   DATA[540,19] := 2.0;
   DATA[540,20] := 148.808;
   DATA[540,21] := 155.9344;
   DATA[540,22] := 1.72095;
   DATA[540,23] := 983.6708;
   DATA[540,24] := 2.0;
   DATA[540,25] := 2.0;
   DATA[540,26] := 7.880544;
   DATA[540,27] := 144.9628;
   DATA[540,28] := 263.4581;
   DATA[540,29] := 12.07383;
   DATA[540,30] := 1.73071;
   DATA[540,31] := 1.275778;
   DATA[540,32] := 0.7353967;
   DATA[540,33] := 0.3065689;
   DATA[540,34] := 2.0;
   DATA[540,35] := 251.0254;
   DATA[540,36] := 1.746067;
   DATA[540,37] := 189.8872;
   DATA[540,38] := 0.000128152;
   DATA[540,39] := 1.0;
   DATA[541,0] := 2.535951;
   DATA[541,1] := 533.7197;
   DATA[541,2] := 2.0;
   DATA[541,3] := 2.0;
   DATA[541,4] := 262.1764;
   DATA[541,5] := 8.395475;
   DATA[541,6] := 327.839;
   DATA[541,7] := 2.439753;
   DATA[541,8] := 2.0;
   DATA[541,9] := 2.0;
   DATA[541,10] := 2.0;
   DATA[541,11] := 19.77399;
   DATA[541,12] := 2.214009;
   DATA[541,13] := 980.7582;
   DATA[541,14] := 1.0;
   DATA[541,15] := 2.0;
   DATA[541,16] := 1.0;
   DATA[541,17] := 1.0;
   DATA[541,18] := 1.0;
   DATA[541,19] := 2.0;
   DATA[541,20] := 148.808;
   DATA[541,21] := 155.9344;
   DATA[541,22] := 1.72095;
   DATA[541,23] := 983.7093;
   DATA[541,24] := 2.0;
   DATA[541,25] := 2.0;
   DATA[541,26] := 7.87766;
   DATA[541,27] := 144.9628;
   DATA[541,28] := 263.4581;
   DATA[541,29] := 12.07383;
   DATA[541,30] := 1.730838;
   DATA[541,31] := 1.290893;
   DATA[541,32] := 0.7353967;
   DATA[541,33] := 0.3065689;
   DATA[541,34] := 2.0;
   DATA[541,35] := 251.0254;
   DATA[541,36] := 1.746067;
   DATA[541,37] := 189.8872;
   DATA[541,38] := 0.000128152;
   DATA[541,39] := 1.0;
   DATA[542,0] := 2.51225;
   DATA[542,1] := 534.2693;
   DATA[542,2] := 2.0;
   DATA[542,3] := 2.0;
   DATA[542,4] := 262.1764;
   DATA[542,5] := 8.395475;
   DATA[542,6] := 327.839;
   DATA[542,7] := 2.439753;
   DATA[542,8] := 2.0;
   DATA[542,9] := 2.0;
   DATA[542,10] := 2.0;
   DATA[542,11] := 19.72598;
   DATA[542,12] := 2.214265;
   DATA[542,13] := 980.8783;
   DATA[542,14] := 1.0;
   DATA[542,15] := 2.0;
   DATA[542,16] := 1.0;
   DATA[542,17] := 1.0;
   DATA[542,18] := 1.0;
   DATA[542,19] := 2.0;
   DATA[542,20] := 148.808;
   DATA[542,21] := 155.9344;
   DATA[542,22] := 1.72095;
   DATA[542,23] := 983.9016;
   DATA[542,24] := 2.0;
   DATA[542,25] := 2.0;
   DATA[542,26] := 7.87766;
   DATA[542,27] := 144.9628;
   DATA[542,28] := 263.4581;
   DATA[542,29] := 12.07383;
   DATA[542,30] := 1.730838;
   DATA[542,31] := 1.292686;
   DATA[542,32] := 0.7353967;
   DATA[542,33] := 0.3065689;
   DATA[542,34] := 2.0;
   DATA[542,35] := 251.0254;
   DATA[542,36] := 1.665972;
   DATA[542,37] := 189.759;
   DATA[542,38] := 0.000128152;
   DATA[542,39] := 1.0;
   DATA[543,0] := 2.500721;
   DATA[543,1] := 534.7403;
   DATA[543,2] := 2.0;
   DATA[543,3] := 2.0;
   DATA[543,4] := 262.1764;
   DATA[543,5] := 8.395475;
   DATA[543,6] := 327.839;
   DATA[543,7] := 2.439753;
   DATA[543,8] := 2.0;
   DATA[543,9] := 2.0;
   DATA[543,10] := 2.0;
   DATA[543,11] := 19.72598;
   DATA[543,12] := 2.2126;
   DATA[543,13] := 981.1587;
   DATA[543,14] := 1.0;
   DATA[543,15] := 2.0;
   DATA[543,16] := 1.0;
   DATA[543,17] := 1.0;
   DATA[543,18] := 1.0;
   DATA[543,19] := 2.0;
   DATA[543,20] := 148.808;
   DATA[543,21] := 155.9344;
   DATA[543,22] := 1.718002;
   DATA[543,23] := 984.5552;
   DATA[543,24] := 2.0;
   DATA[543,25] := 2.0;
   DATA[543,26] := 7.87766;
   DATA[543,27] := 144.6296;
   DATA[543,28] := 263.4581;
   DATA[543,29] := 12.07383;
   DATA[543,30] := 1.730838;
   DATA[543,31] := 1.292686;
   DATA[543,32] := 0.7353967;
   DATA[543,33] := 0.3065689;
   DATA[543,34] := 2.0;
   DATA[543,35] := 250.8972;
   DATA[543,36] := 1.665972;
   DATA[543,37] := 189.6469;
   DATA[543,38] := 0.000128152;
   DATA[543,39] := 1.0;
   DATA[544,0] := 2.481504;
   DATA[544,1] := 534.6226;
   DATA[544,2] := 2.0;
   DATA[544,3] := 2.0;
   DATA[544,4] := 262.1764;
   DATA[544,5] := 8.395475;
   DATA[544,6] := 327.839;
   DATA[544,7] := 2.441034;
   DATA[544,8] := 2.0;
   DATA[544,9] := 2.0;
   DATA[544,10] := 2.0;
   DATA[544,11] := 19.68756;
   DATA[544,12] := 2.212087;
   DATA[544,13] := 981.1587;
   DATA[544,14] := 1.0;
   DATA[544,15] := 2.0;
   DATA[544,16] := 1.0;
   DATA[544,17] := 1.0;
   DATA[544,18] := 1.0;
   DATA[544,19] := 2.0;
   DATA[544,20] := 148.808;
   DATA[544,21] := 155.9344;
   DATA[544,22] := 1.715824;
   DATA[544,23] := 984.9782;
   DATA[544,24] := 2.0;
   DATA[544,25] := 2.0;
   DATA[544,26] := 7.87766;
   DATA[544,27] := 144.6296;
   DATA[544,28] := 263.4581;
   DATA[544,29] := 12.07383;
   DATA[544,30] := 1.728531;
   DATA[544,31] := 1.292686;
   DATA[544,32] := 0.7353967;
   DATA[544,33] := 0.3065689;
   DATA[544,34] := 2.0;
   DATA[544,35] := 250.8972;
   DATA[544,36] := 1.665972;
   DATA[544,37] := 189.6469;
   DATA[544,38] := 0.000128152;
   DATA[544,39] := 1.0;
   DATA[545,0] := 2.458764;
   DATA[545,1] := 534.6226;
   DATA[545,2] := 2.0;
   DATA[545,3] := 2.0;
   DATA[545,4] := 262.1764;
   DATA[545,5] := 8.395475;
   DATA[545,6] := 327.839;
   DATA[545,7] := 2.442188;
   DATA[545,8] := 2.0;
   DATA[545,9] := 2.0;
   DATA[545,10] := 2.0;
   DATA[545,11] := 19.68436;
   DATA[545,12] := 2.210037;
   DATA[545,13] := 980.8783;
   DATA[545,14] := 1.0;
   DATA[545,15] := 2.0;
   DATA[545,16] := 1.0;
   DATA[545,17] := 1.0;
   DATA[545,18] := 1.0;
   DATA[545,19] := 2.0;
   DATA[545,20] := 148.808;
   DATA[545,21] := 155.9344;
   DATA[545,22] := 1.715824;
   DATA[545,23] := 985.4396;
   DATA[545,24] := 2.0;
   DATA[545,25] := 2.0;
   DATA[545,26] := 7.87766;
   DATA[545,27] := 144.6296;
   DATA[545,28] := 263.4581;
   DATA[545,29] := 12.07383;
   DATA[545,30] := 1.728531;
   DATA[545,31] := 1.292686;
   DATA[545,32] := 0.7353967;
   DATA[545,33] := 0.3065689;
   DATA[545,34] := 2.0;
   DATA[545,35] := 250.8972;
   DATA[545,36] := 1.665972;
   DATA[545,37] := 189.6469;
   DATA[545,38] := 0.000128152;
   DATA[545,39] := 1.0;
   DATA[546,0] := 2.447875;
   DATA[546,1] := 534.4263;
   DATA[546,2] := 2.0;
   DATA[546,3] := 2.0;
   DATA[546,4] := 262.1764;
   DATA[546,5] := 8.395475;
   DATA[546,6] := 327.839;
   DATA[546,7] := 2.442316;
   DATA[546,8] := 2.0;
   DATA[546,9] := 2.0;
   DATA[546,10] := 2.0;
   DATA[546,11] := 19.67155;
   DATA[546,12] := 2.209397;
   DATA[546,13] := 981.0385;
   DATA[546,14] := 1.0;
   DATA[546,15] := 2.0;
   DATA[546,16] := 1.0;
   DATA[546,17] := 1.0;
   DATA[546,18] := 1.0;
   DATA[546,19] := 2.0;
   DATA[546,20] := 148.808;
   DATA[546,21] := 155.9344;
   DATA[546,22] := 1.71467;
   DATA[546,23] := 985.9011;
   DATA[546,24] := 2.0;
   DATA[546,25] := 2.0;
   DATA[546,26] := 7.87766;
   DATA[546,27] := 144.6296;
   DATA[546,28] := 263.4581;
   DATA[546,29] := 12.07383;
   DATA[546,30] := 1.728531;
   DATA[546,31] := 1.275906;
   DATA[546,32] := 0.7353967;
   DATA[546,33] := 0.3065689;
   DATA[546,34] := 2.0;
   DATA[546,35] := 250.737;
   DATA[546,36] := 1.665972;
   DATA[546,37] := 189.6469;
   DATA[546,38] := 0.000128152;
   DATA[546,39] := 1.0;
   DATA[547,0] := 2.431861;
   DATA[547,1] := 533.7197;
   DATA[547,2] := 2.0;
   DATA[547,3] := 2.0;
   DATA[547,4] := 262.1764;
   DATA[547,5] := 8.395475;
   DATA[547,6] := 327.839;
   DATA[547,7] := 2.442316;
   DATA[547,8] := 2.0;
   DATA[547,9] := 2.0;
   DATA[547,10] := 2.0;
   DATA[547,11] := 19.61073;
   DATA[547,12] := 2.209397;
   DATA[547,13] := 980.8783;
   DATA[547,14] := 1.0;
   DATA[547,15] := 2.0;
   DATA[547,16] := 1.0;
   DATA[547,17] := 1.0;
   DATA[547,18] := 1.0;
   DATA[547,19] := 2.0;
   DATA[547,20] := 148.808;
   DATA[547,21] := 155.9344;
   DATA[547,22] := 1.713389;
   DATA[547,23] := 986.5547;
   DATA[547,24] := 2.0;
   DATA[547,25] := 2.0;
   DATA[547,26] := 7.87766;
   DATA[547,27] := 144.7578;
   DATA[547,28] := 263.4581;
   DATA[547,29] := 12.07383;
   DATA[547,30] := 1.728531;
   DATA[547,31] := 1.27898;
   DATA[547,32] := 0.7353967;
   DATA[547,33] := 0.3086186;
   DATA[547,34] := 2.0;
   DATA[547,35] := 250.721;
   DATA[547,36] := 1.665972;
   DATA[547,37] := 189.5668;
   DATA[547,38] := 0.000128152;
   DATA[547,39] := 1.0;
   DATA[548,0] := 2.422573;
   DATA[548,1] := 533.5627;
   DATA[548,2] := 2.0;
   DATA[548,3] := 2.0;
   DATA[548,4] := 262.1764;
   DATA[548,5] := 8.395475;
   DATA[548,6] := 327.839;
   DATA[548,7] := 2.442316;
   DATA[548,8] := 2.0;
   DATA[548,9] := 2.0;
   DATA[548,10] := 2.0;
   DATA[548,11] := 19.61073;
   DATA[548,12] := 2.209397;
   DATA[548,13] := 980.678;
   DATA[548,14] := 1.0;
   DATA[548,15] := 2.0;
   DATA[548,16] := 1.0;
   DATA[548,17] := 1.0;
   DATA[548,18] := 1.0;
   DATA[548,19] := 2.0;
   DATA[548,20] := 148.808;
   DATA[548,21] := 155.9344;
   DATA[548,22] := 1.713389;
   DATA[548,23] := 986.9777;
   DATA[548,24] := 2.0;
   DATA[548,25] := 2.0;
   DATA[548,26] := 7.87766;
   DATA[548,27] := 144.7578;
   DATA[548,28] := 263.4581;
   DATA[548,29] := 12.07383;
   DATA[548,30] := 1.726865;
   DATA[548,31] := 1.28103;
   DATA[548,32] := 0.7353967;
   DATA[548,33] := 0.3086186;
   DATA[548,34] := 2.0;
   DATA[548,35] := 250.721;
   DATA[548,36] := 1.665972;
   DATA[548,37] := 189.5668;
   DATA[548,38] := 0.000128152;
   DATA[548,39] := 1.0;
   DATA[549,0] := 2.417449;
   DATA[549,1] := 532.5814;
   DATA[549,2] := 2.0;
   DATA[549,3] := 2.0;
   DATA[549,4] := 262.1764;
   DATA[549,5] := 8.395475;
   DATA[549,6] := 327.839;
   DATA[549,7] := 2.442316;
   DATA[549,8] := 2.0;
   DATA[549,9] := 2.0;
   DATA[549,10] := 2.0;
   DATA[549,11] := 19.61073;
   DATA[549,12] := 2.205682;
   DATA[549,13] := 981.4791;
   DATA[549,14] := 1.0;
   DATA[549,15] := 2.0;
   DATA[549,16] := 1.0;
   DATA[549,17] := 1.0;
   DATA[549,18] := 1.0;
   DATA[549,19] := 2.0;
   DATA[549,20] := 148.808;
   DATA[549,21] := 155.9344;
   DATA[549,22] := 1.714029;
   DATA[549,23] := 987.7083;
   DATA[549,24] := 2.0;
   DATA[549,25] := 2.0;
   DATA[549,26] := 7.87766;
   DATA[549,27] := 144.7578;
   DATA[549,28] := 263.4581;
   DATA[549,29] := 12.07383;
   DATA[549,30] := 1.726865;
   DATA[549,31] := 1.285513;
   DATA[549,32] := 0.7353967;
   DATA[549,33] := 0.3075937;
   DATA[549,34] := 2.0;
   DATA[549,35] := 250.721;
   DATA[549,36] := 1.665972;
   DATA[549,37] := 189.5668;
   DATA[549,38] := 0.000128152;
   DATA[549,39] := 1.0;
   DATA[550,0] := 2.417449;
   DATA[550,1] := 532.5814;
   DATA[550,2] := 2.0;
   DATA[550,3] := 2.0;
   DATA[550,4] := 262.1764;
   DATA[550,5] := 8.395475;
   DATA[550,6] := 327.839;
   DATA[550,7] := 2.442316;
   DATA[550,8] := 2.0;
   DATA[550,9] := 2.0;
   DATA[550,10] := 2.0;
   DATA[550,11] := 19.61073;
   DATA[550,12] := 2.205682;
   DATA[550,13] := 981.4791;
   DATA[550,14] := 1.0;
   DATA[550,15] := 2.0;
   DATA[550,16] := 1.0;
   DATA[550,17] := 1.0;
   DATA[550,18] := 1.0;
   DATA[550,19] := 2.0;
   DATA[550,20] := 148.808;
   DATA[550,21] := 155.9344;
   DATA[550,22] := 1.714029;
   DATA[550,23] := 987.7083;
   DATA[550,24] := 2.0;
   DATA[550,25] := 2.0;
   DATA[550,26] := 7.87766;
   DATA[550,27] := 144.7578;
   DATA[550,28] := 263.4581;
   DATA[550,29] := 12.07383;
   DATA[550,30] := 1.726865;
   DATA[550,31] := 1.285513;
   DATA[550,32] := 0.7353967;
   DATA[550,33] := 0.3075937;
   DATA[550,34] := 2.0;
   DATA[550,35] := 250.721;
   DATA[550,36] := 1.665972;
   DATA[550,37] := 189.5668;
   DATA[550,38] := 0.000128152;
   DATA[550,39] := 1.0;
   DATA[551,0] := 2.423534;
   DATA[551,1] := 532.2674;
   DATA[551,2] := 2.0;
   DATA[551,3] := 2.0;
   DATA[551,4] := 262.1764;
   DATA[551,5] := 8.395475;
   DATA[551,6] := 327.839;
   DATA[551,7] := 2.441547;
   DATA[551,8] := 2.0;
   DATA[551,9] := 2.0;
   DATA[551,10] := 2.0;
   DATA[551,11] := 19.61073;
   DATA[551,12] := 2.205682;
   DATA[551,13] := 981.5593;
   DATA[551,14] := 1.0;
   DATA[551,15] := 2.0;
   DATA[551,16] := 1.0;
   DATA[551,17] := 1.0;
   DATA[551,18] := 1.0;
   DATA[551,19] := 2.0;
   DATA[551,20] := 148.808;
   DATA[551,21] := 155.9344;
   DATA[551,22] := 1.716849;
   DATA[551,23] := 988.0159;
   DATA[551,24] := 2.0;
   DATA[551,25] := 2.0;
   DATA[551,26] := 7.87766;
   DATA[551,27] := 144.7578;
   DATA[551,28] := 263.4581;
   DATA[551,29] := 12.07383;
   DATA[551,30] := 1.726865;
   DATA[551,31] := 1.291405;
   DATA[551,32] := 0.7353967;
   DATA[551,33] := 0.3065689;
   DATA[551,34] := 2.0;
   DATA[551,35] := 250.9773;
   DATA[551,36] := 1.665972;
   DATA[551,37] := 189.5668;
   DATA[551,38] := 0.000128152;
   DATA[551,39] := 1.0;
   DATA[552,0] := 2.455241;
   DATA[552,1] := 531.3253;
   DATA[552,2] := 2.0;
   DATA[552,3] := 2.0;
   DATA[552,4] := 262.1764;
   DATA[552,5] := 8.395475;
   DATA[552,6] := 327.839;
   DATA[552,7] := 2.441547;
   DATA[552,8] := 2.0;
   DATA[552,9] := 2.0;
   DATA[552,10] := 2.0;
   DATA[552,11] := 19.67155;
   DATA[552,12] := 2.208884;
   DATA[552,13] := 981.8796;
   DATA[552,14] := 1.0;
   DATA[552,15] := 2.0;
   DATA[552,16] := 1.0;
   DATA[552,17] := 1.0;
   DATA[552,18] := 1.0;
   DATA[552,19] := 2.0;
   DATA[552,20] := 148.808;
   DATA[552,21] := 155.9344;
   DATA[552,22] := 1.718771;
   DATA[552,23] := 987.939;
   DATA[552,24] := 2.0;
   DATA[552,25] := 2.0;
   DATA[552,26] := 7.87766;
   DATA[552,27] := 144.7578;
   DATA[552,28] := 263.4581;
   DATA[552,29] := 12.07383;
   DATA[552,30] := 1.726865;
   DATA[552,31] := 1.28436;
   DATA[552,32] := 0.7377012;
   DATA[552,33] := 0.3062486;
   DATA[552,34] := 2.0;
   DATA[552,35] := 251.0574;
   DATA[552,36] := 1.778105;
   DATA[552,37] := 189.743;
   DATA[552,38] := 0.000128152;
   DATA[552,39] := 1.0;
   DATA[553,0] := 2.494315;
   DATA[553,1] := 530.7758;
   DATA[553,2] := 2.0;
   DATA[553,3] := 2.0;
   DATA[553,4] := 262.1764;
   DATA[553,5] := 8.395475;
   DATA[553,6] := 327.839;
   DATA[553,7] := 2.441547;
   DATA[553,8] := 2.0;
   DATA[553,9] := 2.0;
   DATA[553,10] := 2.0;
   DATA[553,11] := 19.70037;
   DATA[553,12] := 2.208884;
   DATA[553,13] := 981.7595;
   DATA[553,14] := 1.0;
   DATA[553,15] := 2.0;
   DATA[553,16] := 1.0;
   DATA[553,17] := 1.0;
   DATA[553,18] := 1.0;
   DATA[553,19] := 2.0;
   DATA[553,20] := 148.808;
   DATA[553,21] := 155.9344;
   DATA[553,22] := 1.719924;
   DATA[553,23] := 988.2081;
   DATA[553,24] := 2.0;
   DATA[553,25] := 2.0;
   DATA[553,26] := 7.878942;
   DATA[553,27] := 144.7578;
   DATA[553,28] := 263.4581;
   DATA[553,29] := 12.07383;
   DATA[553,30] := 1.726865;
   DATA[553,31] := 1.281542;
   DATA[553,32] := 0.7377012;
   DATA[553,33] := 0.3062486;
   DATA[553,34] := 2.0;
   DATA[553,35] := 251.2016;
   DATA[553,36] := 1.778105;
   DATA[553,37] := 189.8231;
   DATA[553,38] := 0.000128152;
   DATA[553,39] := 1.0;
   DATA[554,0] := 2.54652;
   DATA[554,1] := 529.7159;
   DATA[554,2] := 2.0;
   DATA[554,3] := 2.0;
   DATA[554,4] := 262.1764;
   DATA[554,5] := 8.395475;
   DATA[554,6] := 327.839;
   DATA[554,7] := 2.441547;
   DATA[554,8] := 2.0;
   DATA[554,9] := 2.0;
   DATA[554,10] := 2.0;
   DATA[554,11] := 19.71637;
   DATA[554,12] := 2.208884;
   DATA[554,13] := 981.5593;
   DATA[554,14] := 1.0;
   DATA[554,15] := 2.0;
   DATA[554,16] := 1.0;
   DATA[554,17] := 1.0;
   DATA[554,18] := 1.0;
   DATA[554,19] := 2.0;
   DATA[554,20] := 148.808;
   DATA[554,21] := 155.9344;
   DATA[554,22] := 1.723256;
   DATA[554,23] := 988.5157;
   DATA[554,24] := 2.0;
   DATA[554,25] := 2.0;
   DATA[554,26] := 7.880544;
   DATA[554,27] := 144.7578;
   DATA[554,28] := 263.4581;
   DATA[554,29] := 12.07383;
   DATA[554,30] := 1.726865;
   DATA[554,31] := 1.281542;
   DATA[554,32] := 0.7377012;
   DATA[554,33] := 0.3062486;
   DATA[554,34] := 2.0;
   DATA[554,35] := 251.2977;
   DATA[554,36] := 1.778105;
   DATA[554,37] := 189.9833;
   DATA[554,38] := 0.000128152;
   DATA[554,39] := 1.0;
   DATA[555,0] := 2.570541;
   DATA[555,1] := 529.3627;
   DATA[555,2] := 2.0;
   DATA[555,3] := 2.0;
   DATA[555,4] := 262.1764;
   DATA[555,5] := 8.395475;
   DATA[555,6] := 327.839;
   DATA[555,7] := 2.441547;
   DATA[555,8] := 2.0;
   DATA[555,9] := 2.0;
   DATA[555,10] := 2.0;
   DATA[555,11] := 19.75159;
   DATA[555,12] := 2.208884;
   DATA[555,13] := 981.2789;
   DATA[555,14] := 1.0;
   DATA[555,15] := 2.0;
   DATA[555,16] := 1.0;
   DATA[555,17] := 1.0;
   DATA[555,18] := 1.0;
   DATA[555,19] := 2.0;
   DATA[555,20] := 148.808;
   DATA[555,21] := 155.9344;
   DATA[555,22] := 1.724153;
   DATA[555,23] := 988.4388;
   DATA[555,24] := 2.0;
   DATA[555,25] := 2.0;
   DATA[555,26] := 7.880544;
   DATA[555,27] := 144.7578;
   DATA[555,28] := 263.4581;
   DATA[555,29] := 12.07383;
   DATA[555,30] := 1.728019;
   DATA[555,31] := 1.288715;
   DATA[555,32] := 0.7379573;
   DATA[555,33] := 0.3062486;
   DATA[555,34] := 2.0;
   DATA[555,35] := 251.2977;
   DATA[555,36] := 1.778105;
   DATA[555,37] := 190.0474;
   DATA[555,38] := 0.000128152;
   DATA[555,39] := 1.0;
   DATA[556,0] := 2.61634;
   DATA[556,1] := 528.5776;
   DATA[556,2] := 2.0;
   DATA[556,3] := 2.0;
   DATA[556,4] := 262.1764;
   DATA[556,5] := 8.395475;
   DATA[556,6] := 327.839;
   DATA[556,7] := 2.441547;
   DATA[556,8] := 2.0;
   DATA[556,9] := 2.0;
   DATA[556,10] := 2.0;
   DATA[556,11] := 19.79;
   DATA[556,12] := 2.208372;
   DATA[556,13] := 981.1987;
   DATA[556,14] := 1.0;
   DATA[556,15] := 2.0;
   DATA[556,16] := 1.0;
   DATA[556,17] := 1.0;
   DATA[556,18] := 1.0;
   DATA[556,19] := 2.0;
   DATA[556,20] := 148.808;
   DATA[556,21] := 156.0369;
   DATA[556,22] := 1.724153;
   DATA[556,23] := 989.0156;
   DATA[556,24] := 2.0;
   DATA[556,25] := 2.0;
   DATA[556,26] := 7.880544;
   DATA[556,27] := 144.7578;
   DATA[556,28] := 263.4581;
   DATA[556,29] := 12.07383;
   DATA[556,30] := 1.729172;
   DATA[556,31] := 1.292558;
   DATA[556,32] := 0.7357808;
   DATA[556,33] := 0.3066329;
   DATA[556,34] := 2.0;
   DATA[556,35] := 251.2977;
   DATA[556,36] := 1.778105;
   DATA[556,37] := 190.0474;
   DATA[556,38] := 0.000128152;
   DATA[556,39] := 1.0;
   DATA[557,0] := 2.641322;
   DATA[557,1] := 528.4599;
   DATA[557,2] := 2.0;
   DATA[557,3] := 2.0;
   DATA[557,4] := 262.1764;
   DATA[557,5] := 8.395475;
   DATA[557,6] := 327.9159;
   DATA[557,7] := 2.441162;
   DATA[557,8] := 2.0;
   DATA[557,9] := 2.0;
   DATA[557,10] := 2.0;
   DATA[557,11] := 19.80601;
   DATA[557,12] := 2.208372;
   DATA[557,13] := 981.4391;
   DATA[557,14] := 1.0;
   DATA[557,15] := 2.0;
   DATA[557,16] := 1.0;
   DATA[557,17] := 1.0;
   DATA[557,18] := 1.0;
   DATA[557,19] := 2.0;
   DATA[557,20] := 148.808;
   DATA[557,21] := 156.0369;
   DATA[557,22] := 1.724153;
   DATA[557,23] := 988.708;
   DATA[557,24] := 2.0;
   DATA[557,25] := 2.0;
   DATA[557,26] := 7.880544;
   DATA[557,27] := 144.7578;
   DATA[557,28] := 263.4581;
   DATA[557,29] := 12.07383;
   DATA[557,30] := 1.729172;
   DATA[557,31] := 1.292558;
   DATA[557,32] := 0.7357808;
   DATA[557,33] := 0.3066329;
   DATA[557,34] := 2.0;
   DATA[557,35] := 251.2977;
   DATA[557,36] := 1.778105;
   DATA[557,37] := 190.0474;
   DATA[557,38] := 0.000128152;
   DATA[557,39] := 1.0;
   DATA[558,0] := 2.672389;
   DATA[558,1] := 528.8132;
   DATA[558,2] := 2.0;
   DATA[558,3] := 2.0;
   DATA[558,4] := 262.1764;
   DATA[558,5] := 8.395475;
   DATA[558,6] := 327.9159;
   DATA[558,7] := 2.440265;
   DATA[558,8] := 2.0;
   DATA[558,9] := 2.0;
   DATA[558,10] := 2.0;
   DATA[558,11] := 19.80601;
   DATA[558,12] := 2.210806;
   DATA[558,13] := 981.7996;
   DATA[558,14] := 1.0;
   DATA[558,15] := 2.0;
   DATA[558,16] := 1.0;
   DATA[558,17] := 1.0;
   DATA[558,18] := 1.0;
   DATA[558,19] := 2.0;
   DATA[558,20] := 148.808;
   DATA[558,21] := 156.0369;
   DATA[558,22] := 1.724153;
   DATA[558,23] := 988.9003;
   DATA[558,24] := 2.0;
   DATA[558,25] := 2.0;
   DATA[558,26] := 7.880544;
   DATA[558,27] := 144.7578;
   DATA[558,28] := 263.4581;
   DATA[558,29] := 12.07383;
   DATA[558,30] := 1.729172;
   DATA[558,31] := 1.292174;
   DATA[558,32] := 0.7357808;
   DATA[558,33] := 0.3074656;
   DATA[558,34] := 2.0;
   DATA[558,35] := 251.2977;
   DATA[558,36] := 1.778105;
   DATA[558,37] := 190.0474;
   DATA[558,38] := 0.000128152;
   DATA[558,39] := 1.0;
   DATA[559,0] := 2.674951;
   DATA[559,1] := 528.7739;
   DATA[559,2] := 2.0;
   DATA[559,3] := 2.0;
   DATA[559,4] := 262.1764;
   DATA[559,5] := 8.395475;
   DATA[559,6] := 327.9159;
   DATA[559,7] := 2.440265;
   DATA[559,8] := 2.0;
   DATA[559,9] := 2.0;
   DATA[559,10] := 2.0;
   DATA[559,11] := 19.73238;
   DATA[559,12] := 2.211959;
   DATA[559,13] := 981.5993;
   DATA[559,14] := 1.0;
   DATA[559,15] := 2.0;
   DATA[559,16] := 1.0;
   DATA[559,17] := 1.0;
   DATA[559,18] := 1.0;
   DATA[559,19] := 2.0;
   DATA[559,20] := 148.808;
   DATA[559,21] := 156.0369;
   DATA[559,22] := 1.723641;
   DATA[559,23] := 988.6696;
   DATA[559,24] := 2.0;
   DATA[559,25] := 2.0;
   DATA[559,26] := 7.880544;
   DATA[559,27] := 144.7578;
   DATA[559,28] := 263.4581;
   DATA[559,29] := 12.07383;
   DATA[559,30] := 1.730838;
   DATA[559,31] := 1.283079;
   DATA[559,32] := 0.7353967;
   DATA[559,33] := 0.3080421;
   DATA[559,34] := 2.0;
   DATA[559,35] := 251.2977;
   DATA[559,36] := 1.746067;
   DATA[559,37] := 190.0474;
   DATA[559,38] := 0.000128152;
   DATA[559,39] := 1.0;
   DATA[560,0] := 2.643244;
   DATA[560,1] := 529.6375;
   DATA[560,2] := 2.0;
   DATA[560,3] := 2.0;
   DATA[560,4] := 262.1764;
   DATA[560,5] := 8.395475;
   DATA[560,6] := 327.9159;
   DATA[560,7] := 2.4427;
   DATA[560,8] := 2.0;
   DATA[560,9] := 2.0;
   DATA[560,10] := 2.0;
   DATA[560,11] := 19.69076;
   DATA[560,12] := 2.211959;
   DATA[560,13] := 981.1987;
   DATA[560,14] := 1.0;
   DATA[560,15] := 2.0;
   DATA[560,16] := 1.0;
   DATA[560,17] := 1.0;
   DATA[560,18] := 1.0;
   DATA[560,19] := 2.0;
   DATA[560,20] := 148.808;
   DATA[560,21] := 156.0369;
   DATA[560,22] := 1.722487;
   DATA[560,23] := 988.6696;
   DATA[560,24] := 2.0;
   DATA[560,25] := 2.0;
   DATA[560,26] := 7.880544;
   DATA[560,27] := 144.7578;
   DATA[560,28] := 263.4581;
   DATA[560,29] := 12.07383;
   DATA[560,30] := 1.731479;
   DATA[560,31] := 1.287306;
   DATA[560,32] := 0.7353967;
   DATA[560,33] := 0.3080421;
   DATA[560,34] := 2.0;
   DATA[560,35] := 251.2977;
   DATA[560,36] := 1.746067;
   DATA[560,37] := 190.0474;
   DATA[560,38] := 0.000128152;
   DATA[560,39] := 1.0;
   DATA[561,0] := 2.621785;
   DATA[561,1] := 530.344;
   DATA[561,2] := 2.0;
   DATA[561,3] := 2.0;
   DATA[561,4] := 262.1764;
   DATA[561,5] := 8.395475;
   DATA[561,6] := 327.9159;
   DATA[561,7] := 2.4427;
   DATA[561,8] := 2.0;
   DATA[561,9] := 2.0;
   DATA[561,10] := 2.0;
   DATA[561,11] := 19.66835;
   DATA[561,12] := 2.211959;
   DATA[561,13] := 981.4791;
   DATA[561,14] := 1.0;
   DATA[561,15] := 2.0;
   DATA[561,16] := 1.0;
   DATA[561,17] := 1.0;
   DATA[561,18] := 1.0;
   DATA[561,19] := 2.0;
   DATA[561,20] := 148.808;
   DATA[561,21] := 156.0369;
   DATA[561,22] := 1.72159;
   DATA[561,23] := 988.7465;
   DATA[561,24] := 2.0;
   DATA[561,25] := 2.0;
   DATA[561,26] := 7.880544;
   DATA[561,27] := 144.7578;
   DATA[561,28] := 263.4261;
   DATA[561,29] := 12.07383;
   DATA[561,30] := 1.731479;
   DATA[561,31] := 1.274625;
   DATA[561,32] := 0.7353967;
   DATA[561,33] := 0.3087468;
   DATA[561,34] := 2.0;
   DATA[561,35] := 251.2977;
   DATA[561,36] := 1.746067;
   DATA[561,37] := 190.0474;
   DATA[561,38] := 0.000128152;
   DATA[561,39] := 1.0;
   DATA[562,0] := 2.61634;
   DATA[562,1] := 531.9534;
   DATA[562,2] := 2.0;
   DATA[562,3] := 2.0;
   DATA[562,4] := 262.1764;
   DATA[562,5] := 8.395475;
   DATA[562,6] := 327.9159;
   DATA[562,7] := 2.4427;
   DATA[562,8] := 2.0;
   DATA[562,9] := 2.0;
   DATA[562,10] := 2.0;
   DATA[562,11] := 19.66835;
   DATA[562,12] := 2.214906;
   DATA[562,13] := 981.4391;
   DATA[562,14] := 1.0;
   DATA[562,15] := 2.0;
   DATA[562,16] := 1.0;
   DATA[562,17] := 1.0;
   DATA[562,18] := 1.0;
   DATA[562,19] := 2.0;
   DATA[562,20] := 148.808;
   DATA[562,21] := 156.0369;
   DATA[562,22] := 1.718515;
   DATA[562,23] := 989.0925;
   DATA[562,24] := 2.0;
   DATA[562,25] := 2.0;
   DATA[562,26] := 7.880544;
   DATA[562,27] := 144.7578;
   DATA[562,28] := 263.4261;
   DATA[562,29] := 12.07383;
   DATA[562,30] := 1.731479;
   DATA[562,31] := 1.261432;
   DATA[562,32] := 0.7353967;
   DATA[562,33] := 0.3068891;
   DATA[562,34] := 2.0;
   DATA[562,35] := 251.0734;
   DATA[562,36] := 1.746067;
   DATA[562,37] := 189.727;
   DATA[562,38] := 0.000128152;
   DATA[562,39] := 1.0;
   DATA[563,0] := 2.6157;
   DATA[563,1] := 532.5422;
   DATA[563,2] := 2.0;
   DATA[563,3] := 2.0;
   DATA[563,4] := 262.1764;
   DATA[563,5] := 8.395155;
   DATA[563,6] := 327.9159;
   DATA[563,7] := 2.4427;
   DATA[563,8] := 2.0;
   DATA[563,9] := 2.0;
   DATA[563,10] := 2.0;
   DATA[563,11] := 19.66835;
   DATA[563,12] := 2.214906;
   DATA[563,13] := 981.5593;
   DATA[563,14] := 1.0;
   DATA[563,15] := 2.0;
   DATA[563,16] := 1.0;
   DATA[563,17] := 1.0;
   DATA[563,18] := 1.0;
   DATA[563,19] := 2.0;
   DATA[563,20] := 148.808;
   DATA[563,21] := 156.0369;
   DATA[563,22] := 1.718515;
   DATA[563,23] := 988.708;
   DATA[563,24] := 2.0;
   DATA[563,25] := 2.0;
   DATA[563,26] := 7.880544;
   DATA[563,27] := 144.7578;
   DATA[563,28] := 263.4261;
   DATA[563,29] := 12.07383;
   DATA[563,30] := 1.731479;
   DATA[563,31] := 1.25554;
   DATA[563,32] := 0.7353967;
   DATA[563,33] := 0.3066329;
   DATA[563,34] := 2.0;
   DATA[563,35] := 251.0734;
   DATA[563,36] := 1.746067;
   DATA[563,37] := 189.727;
   DATA[563,38] := 0.000128152;
   DATA[563,39] := 1.0;
   DATA[564,0] := 2.593601;
   DATA[564,1] := 532.8954;
   DATA[564,2] := 2.0;
   DATA[564,3] := 2.0;
   DATA[564,4] := 262.1764;
   DATA[564,5] := 8.394835;
   DATA[564,6] := 327.9159;
   DATA[564,7] := 2.444879;
   DATA[564,8] := 2.0;
   DATA[564,9] := 2.0;
   DATA[564,10] := 2.0;
   DATA[564,11] := 19.66835;
   DATA[564,12] := 2.21324;
   DATA[564,13] := 980.8383;
   DATA[564,14] := 1.0;
   DATA[564,15] := 2.0;
   DATA[564,16] := 1.0;
   DATA[564,17] := 1.0;
   DATA[564,18] := 1.0;
   DATA[564,19] := 2.0;
   DATA[564,20] := 148.808;
   DATA[564,21] := 156.0369;
   DATA[564,22] := 1.718515;
   DATA[564,23] := 989.0925;
   DATA[564,24] := 2.0;
   DATA[564,25] := 2.0;
   DATA[564,26] := 7.880544;
   DATA[564,27] := 144.7578;
   DATA[564,28] := 263.4261;
   DATA[564,29] := 12.07383;
   DATA[564,30] := 1.7293;
   DATA[564,31] := 1.254643;
   DATA[564,32] := 0.7353967;
   DATA[564,33] := 0.3065048;
   DATA[564,34] := 2.0;
   DATA[564,35] := 250.9773;
   DATA[564,36] := 1.746067;
   DATA[564,37] := 189.727;
   DATA[564,38] := 0.000128152;
   DATA[564,39] := 1.0;
   DATA[565,0] := 2.572142;
   DATA[565,1] := 532.9739;
   DATA[565,2] := 2.0;
   DATA[565,3] := 2.0;
   DATA[565,4] := 262.1764;
   DATA[565,5] := 8.394835;
   DATA[565,6] := 327.9159;
   DATA[565,7] := 2.444879;
   DATA[565,8] := 2.0;
   DATA[565,9] := 2.0;
   DATA[565,10] := 2.0;
   DATA[565,11] := 19.67796;
   DATA[565,12] := 2.21324;
   DATA[565,13] := 981.1587;
   DATA[565,14] := 1.0;
   DATA[565,15] := 2.0;
   DATA[565,16] := 1.0;
   DATA[565,17] := 1.0;
   DATA[565,18] := 1.0;
   DATA[565,19] := 2.0;
   DATA[565,20] := 148.808;
   DATA[565,21] := 156.0369;
   DATA[565,22] := 1.718515;
   DATA[565,23] := 988.9387;
   DATA[565,24] := 2.0;
   DATA[565,25] := 2.0;
   DATA[565,26] := 7.880544;
   DATA[565,27] := 144.7578;
   DATA[565,28] := 263.4261;
   DATA[565,29] := 12.07383;
   DATA[565,30] := 1.7293;
   DATA[565,31] := 1.268989;
   DATA[565,32] := 0.7353967;
   DATA[565,33] := 0.3065048;
   DATA[565,34] := 2.0;
   DATA[565,35] := 250.9132;
   DATA[565,36] := 1.746067;
   DATA[565,37] := 189.5988;
   DATA[565,38] := 0.000128152;
   DATA[565,39] := 1.0;
   DATA[566,0] := 2.560933;
   DATA[566,1] := 532.8562;
   DATA[566,2] := 2.0;
   DATA[566,3] := 2.0;
   DATA[566,4] := 262.1764;
   DATA[566,5] := 8.394835;
   DATA[566,6] := 327.9159;
   DATA[566,7] := 2.444879;
   DATA[566,8] := 2.0;
   DATA[566,9] := 2.0;
   DATA[566,10] := 2.0;
   DATA[566,11] := 19.67796;
   DATA[566,12] := 2.21324;
   DATA[566,13] := 981.1987;
   DATA[566,14] := 1.0;
   DATA[566,15] := 2.0;
   DATA[566,16] := 1.0;
   DATA[566,17] := 1.0;
   DATA[566,18] := 1.0;
   DATA[566,19] := 2.0;
   DATA[566,20] := 148.808;
   DATA[566,21] := 156.0369;
   DATA[566,22] := 1.717105;
   DATA[566,23] := 988.4773;
   DATA[566,24] := 2.0;
   DATA[566,25] := 2.0;
   DATA[566,26] := 7.880544;
   DATA[566,27] := 144.7578;
   DATA[566,28] := 263.4261;
   DATA[566,29] := 12.07383;
   DATA[566,30] := 1.726096;
   DATA[566,31] := 1.271039;
   DATA[566,32] := 0.736421;
   DATA[566,33] := 0.3065048;
   DATA[566,34] := 2.0;
   DATA[566,35] := 250.5928;
   DATA[566,36] := 1.665972;
   DATA[566,37] := 189.5347;
   DATA[566,38] := 0.000128152;
   DATA[566,39] := 1.0;
   DATA[567,0] := 2.542036;
   DATA[567,1] := 532.7384;
   DATA[567,2] := 2.0;
   DATA[567,3] := 2.0;
   DATA[567,4] := 262.1764;
   DATA[567,5] := 8.394835;
   DATA[567,6] := 327.9159;
   DATA[567,7] := 2.442444;
   DATA[567,8] := 2.0;
   DATA[567,9] := 2.0;
   DATA[567,10] := 2.0;
   DATA[567,11] := 19.67796;
   DATA[567,12] := 2.21324;
   DATA[567,13] := 981.1587;
   DATA[567,14] := 1.0;
   DATA[567,15] := 2.0;
   DATA[567,16] := 1.0;
   DATA[567,17] := 1.0;
   DATA[567,18] := 1.0;
   DATA[567,19] := 2.0;
   DATA[567,20] := 148.808;
   DATA[567,21] := 156.0369;
   DATA[567,22] := 1.716592;
   DATA[567,23] := 989.0541;
   DATA[567,24] := 2.0;
   DATA[567,25] := 2.0;
   DATA[567,26] := 7.880544;
   DATA[567,27] := 144.8859;
   DATA[567,28] := 263.4261;
   DATA[567,29] := 12.07383;
   DATA[567,30] := 1.726096;
   DATA[567,31] := 1.280261;
   DATA[567,32] := 0.7370611;
   DATA[567,33] := 0.3065048;
   DATA[567,34] := 2.0;
   DATA[567,35] := 250.5928;
   DATA[567,36] := 1.665972;
   DATA[567,37] := 189.5027;
   DATA[567,38] := 0.000128152;
   DATA[567,39] := 1.0;
   DATA[568,0] := 2.530506;
   DATA[568,1] := 532.4637;
   DATA[568,2] := 2.0;
   DATA[568,3] := 2.0;
   DATA[568,4] := 262.1764;
   DATA[568,5] := 8.394835;
   DATA[568,6] := 327.9159;
   DATA[568,7] := 2.441162;
   DATA[568,8] := 2.0;
   DATA[568,9] := 2.0;
   DATA[568,10] := 2.0;
   DATA[568,11] := 19.63954;
   DATA[568,12] := 2.211318;
   DATA[568,13] := 980.9985;
   DATA[568,14] := 1.0;
   DATA[568,15] := 2.0;
   DATA[568,16] := 1.0;
   DATA[568,17] := 1.0;
   DATA[568,18] := 1.0;
   DATA[568,19] := 2.0;
   DATA[568,20] := 148.808;
   DATA[568,21] := 156.0369;
   DATA[568,22] := 1.716592;
   DATA[568,23] := 988.708;
   DATA[568,24] := 2.0;
   DATA[568,25] := 2.0;
   DATA[568,26] := 7.880544;
   DATA[568,27] := 144.9116;
   DATA[568,28] := 263.4261;
   DATA[568,29] := 12.07383;
   DATA[568,30] := 1.726096;
   DATA[568,31] := 1.290124;
   DATA[568,32] := 0.7370611;
   DATA[568,33] := 0.3083624;
   DATA[568,34] := 2.0;
   DATA[568,35] := 250.5928;
   DATA[568,36] := 1.665972;
   DATA[568,37] := 189.5027;
   DATA[568,38] := 0.000128152;
   DATA[568,39] := 1.0;
   DATA[569,0] := 2.510649;
   DATA[569,1] := 532.2674;
   DATA[569,2] := 2.0;
   DATA[569,3] := 2.0;
   DATA[569,4] := 262.1764;
   DATA[569,5] := 8.394835;
   DATA[569,6] := 327.9159;
   DATA[569,7] := 2.440521;
   DATA[569,8] := 2.0;
   DATA[569,9] := 2.0;
   DATA[569,10] := 2.0;
   DATA[569,11] := 19.63954;
   DATA[569,12] := 2.210294;
   DATA[569,13] := 980.638;
   DATA[569,14] := 1.0;
   DATA[569,15] := 2.0;
   DATA[569,16] := 1.0;
   DATA[569,17] := 1.0;
   DATA[569,18] := 1.0;
   DATA[569,19] := 2.0;
   DATA[569,20] := 148.808;
   DATA[569,21] := 156.0369;
   DATA[569,22] := 1.717746;
   DATA[569,23] := 988.8618;
   DATA[569,24] := 2.0;
   DATA[569,25] := 2.0;
   DATA[569,26] := 7.880544;
   DATA[569,27] := 144.9116;
   DATA[569,28] := 263.4261;
   DATA[569,29] := 12.07383;
   DATA[569,30] := 1.726096;
   DATA[569,31] := 1.291277;
   DATA[569,32] := 0.7370611;
   DATA[569,33] := 0.3083624;
   DATA[569,34] := 2.0;
   DATA[569,35] := 250.8171;
   DATA[569,36] := 1.665972;
   DATA[569,37] := 189.5027;
   DATA[569,38] := 0.000128152;
   DATA[569,39] := 1.0;
   DATA[570,0] := 2.498799;
   DATA[570,1] := 532.3459;
   DATA[570,2] := 2.0;
   DATA[570,3] := 2.0;
   DATA[570,4] := 262.1764;
   DATA[570,5] := 8.394835;
   DATA[570,6] := 327.9159;
   DATA[570,7] := 2.439881;
   DATA[570,8] := 2.0;
   DATA[570,9] := 2.0;
   DATA[570,10] := 2.0;
   DATA[570,11] := 19.63954;
   DATA[570,12] := 2.210294;
   DATA[570,13] := 980.598;
   DATA[570,14] := 1.0;
   DATA[570,15] := 2.0;
   DATA[570,16] := 1.0;
   DATA[570,17] := 1.0;
   DATA[570,18] := 1.0;
   DATA[570,19] := 2.0;
   DATA[570,20] := 148.808;
   DATA[570,21] := 156.0369;
   DATA[570,22] := 1.717746;
   DATA[570,23] := 988.8618;
   DATA[570,24] := 2.0;
   DATA[570,25] := 2.0;
   DATA[570,26] := 7.880544;
   DATA[570,27] := 144.9116;
   DATA[570,28] := 263.4261;
   DATA[570,29] := 12.07383;
   DATA[570,30] := 1.726096;
   DATA[570,31] := 1.286025;
   DATA[570,32] := 0.7359089;
   DATA[570,33] := 0.3083624;
   DATA[570,34] := 2.0;
   DATA[570,35] := 250.8652;
   DATA[570,36] := 1.665972;
   DATA[570,37] := 189.5027;
   DATA[570,38] := 0.000128152;
   DATA[570,39] := 1.0;
   DATA[571,0] := 2.484066;
   DATA[571,1] := 532.1497;
   DATA[571,2] := 2.0;
   DATA[571,3] := 2.0;
   DATA[571,4] := 262.1764;
   DATA[571,5] := 8.394835;
   DATA[571,6] := 327.9159;
   DATA[571,7] := 2.439881;
   DATA[571,8] := 2.0;
   DATA[571,9] := 2.0;
   DATA[571,10] := 2.0;
   DATA[571,11] := 19.65875;
   DATA[571,12] := 2.214777;
   DATA[571,13] := 980.638;
   DATA[571,14] := 1.0;
   DATA[571,15] := 2.0;
   DATA[571,16] := 1.0;
   DATA[571,17] := 1.0;
   DATA[571,18] := 1.0;
   DATA[571,19] := 2.0;
   DATA[571,20] := 148.808;
   DATA[571,21] := 156.0369;
   DATA[571,22] := 1.717746;
   DATA[571,23] := 989.4386;
   DATA[571,24] := 2.0;
   DATA[571,25] := 2.0;
   DATA[571,26] := 7.880544;
   DATA[571,27] := 144.9116;
   DATA[571,28] := 263.4261;
   DATA[571,29] := 12.07383;
   DATA[571,30] := 1.726096;
   DATA[571,31] := 1.287947;
   DATA[571,32] := 0.7347566;
   DATA[571,33] := 0.3083624;
   DATA[571,34] := 2.0;
   DATA[571,35] := 250.9453;
   DATA[571,36] := 1.665972;
   DATA[571,37] := 189.743;
   DATA[571,38] := 0.000128152;
   DATA[571,39] := 1.0;
   DATA[572,0] := 2.475098;
   DATA[572,1] := 532.0711;
   DATA[572,2] := 2.0;
   DATA[572,3] := 2.0;
   DATA[572,4] := 262.1764;
   DATA[572,5] := 8.394835;
   DATA[572,6] := 327.9159;
   DATA[572,7] := 2.439881;
   DATA[572,8] := 2.0;
   DATA[572,9] := 2.0;
   DATA[572,10] := 2.0;
   DATA[572,11] := 19.65875;
   DATA[572,12] := 2.214777;
   DATA[572,13] := 980.5579;
   DATA[572,14] := 1.0;
   DATA[572,15] := 2.0;
   DATA[572,16] := 1.0;
   DATA[572,17] := 1.0;
   DATA[572,18] := 1.0;
   DATA[572,19] := 2.0;
   DATA[572,20] := 148.808;
   DATA[572,21] := 155.8575;
   DATA[572,22] := 1.717746;
   DATA[572,23] := 989.131;
   DATA[572,24] := 2.0;
   DATA[572,25] := 2.0;
   DATA[572,26] := 7.880544;
   DATA[572,27] := 144.9116;
   DATA[572,28] := 263.4261;
   DATA[572,29] := 12.07383;
   DATA[572,30] := 1.726352;
   DATA[572,31] := 1.272064;
   DATA[572,32] := 0.7347566;
   DATA[572,33] := 0.3083624;
   DATA[572,34] := 2.0;
   DATA[572,35] := 250.9453;
   DATA[572,36] := 1.665972;
   DATA[572,37] := 189.743;
   DATA[572,38] := 0.000128152;
   DATA[572,39] := 1.0;
   DATA[573,0] := 2.462287;
   DATA[573,1] := 531.7964;
   DATA[573,2] := 2.0;
   DATA[573,3] := 2.0;
   DATA[573,4] := 262.1764;
   DATA[573,5] := 8.394835;
   DATA[573,6] := 327.9159;
   DATA[573,7] := 2.439881;
   DATA[573,8] := 2.0;
   DATA[573,9] := 2.0;
   DATA[573,10] := 2.0;
   DATA[573,11] := 19.70037;
   DATA[573,12] := 2.21324;
   DATA[573,13] := 980.7982;
   DATA[573,14] := 1.0;
   DATA[573,15] := 2.0;
   DATA[573,16] := 1.0;
   DATA[573,17] := 1.0;
   DATA[573,18] := 1.0;
   DATA[573,19] := 2.0;
   DATA[573,20] := 148.808;
   DATA[573,21] := 155.8575;
   DATA[573,22] := 1.717746;
   DATA[573,23] := 989.4001;
   DATA[573,24] := 2.0;
   DATA[573,25] := 2.0;
   DATA[573,26] := 7.880544;
   DATA[573,27] := 144.9116;
   DATA[573,28] := 263.4261;
   DATA[573,29] := 12.07383;
   DATA[573,30] := 1.726737;
   DATA[573,31] := 1.280005;
   DATA[573,32] := 0.7347566;
   DATA[573,33] := 0.3083624;
   DATA[573,34] := 2.0;
   DATA[573,35] := 250.9453;
   DATA[573,36] := 1.665972;
   DATA[573,37] := 189.743;
   DATA[573,38] := 0.000128152;
   DATA[573,39] := 1.0;
   DATA[574,0] := 2.449476;
   DATA[574,1] := 531.9141;
   DATA[574,2] := 2.0;
   DATA[574,3] := 2.0;
   DATA[574,4] := 262.1764;
   DATA[574,5] := 8.394835;
   DATA[574,6] := 327.839;
   DATA[574,7] := 2.442188;
   DATA[574,8] := 2.0;
   DATA[574,9] := 2.0;
   DATA[574,10] := 2.0;
   DATA[574,11] := 19.70037;
   DATA[574,12] := 2.212215;
   DATA[574,13] := 980.7982;
   DATA[574,14] := 1.0;
   DATA[574,15] := 2.0;
   DATA[574,16] := 1.0;
   DATA[574,17] := 1.0;
   DATA[574,18] := 1.0;
   DATA[574,19] := 2.0;
   DATA[574,20] := 148.808;
   DATA[574,21] := 155.8575;
   DATA[574,22] := 1.717746;
   DATA[574,23] := 989.3232;
   DATA[574,24] := 2.0;
   DATA[574,25] := 2.0;
   DATA[574,26] := 7.880544;
   DATA[574,27] := 144.9116;
   DATA[574,28] := 263.4261;
   DATA[574,29] := 12.07383;
   DATA[574,30] := 1.726737;
   DATA[574,31] := 1.291405;
   DATA[574,32] := 0.7347566;
   DATA[574,33] := 0.3083624;
   DATA[574,34] := 2.0;
   DATA[574,35] := 250.9453;
   DATA[574,36] := 1.665972;
   DATA[574,37] := 189.743;
   DATA[574,38] := 0.000128152;
   DATA[574,39] := 1.0;
   DATA[575,0] := 2.433142;
   DATA[575,1] := 532.1889;
   DATA[575,2] := 2.0;
   DATA[575,3] := 2.0;
   DATA[575,4] := 262.1764;
   DATA[575,5] := 8.394835;
   DATA[575,6] := 327.839;
   DATA[575,7] := 2.442188;
   DATA[575,8] := 2.0;
   DATA[575,9] := 2.0;
   DATA[575,10] := 2.0;
   DATA[575,11] := 19.73878;
   DATA[575,12] := 2.212215;
   DATA[575,13] := 980.678;
   DATA[575,14] := 1.0;
   DATA[575,15] := 2.0;
   DATA[575,16] := 1.0;
   DATA[575,17] := 1.0;
   DATA[575,18] := 1.0;
   DATA[575,19] := 2.0;
   DATA[575,20] := 148.808;
   DATA[575,21] := 155.678;
   DATA[575,22] := 1.717746;
   DATA[575,23] := 989.4771;
   DATA[575,24] := 2.0;
   DATA[575,25] := 2.0;
   DATA[575,26] := 7.880544;
   DATA[575,27] := 144.9116;
   DATA[575,28] := 263.4261;
   DATA[575,29] := 12.07383;
   DATA[575,30] := 1.728531;
   DATA[575,31] := 1.291405;
   DATA[575,32] := 0.7355248;
   DATA[575,33] := 0.3083624;
   DATA[575,34] := 2.0;
   DATA[575,35] := 250.9773;
   DATA[575,36] := 1.665972;
   DATA[575,37] := 189.743;
   DATA[575,38] := 0.000128152;
   DATA[575,39] := 1.0;
   DATA[576,0] := 2.428979;
   DATA[576,1] := 532.3459;
   DATA[576,2] := 2.0;
   DATA[576,3] := 2.0;
   DATA[576,4] := 262.1764;
   DATA[576,5] := 8.394835;
   DATA[576,6] := 327.839;
   DATA[576,7] := 2.442188;
   DATA[576,8] := 2.0;
   DATA[576,9] := 2.0;
   DATA[576,10] := 2.0;
   DATA[576,11] := 19.74838;
   DATA[576,12] := 2.21055;
   DATA[576,13] := 980.598;
   DATA[576,14] := 1.0;
   DATA[576,15] := 2.0;
   DATA[576,16] := 1.0;
   DATA[576,17] := 1.0;
   DATA[576,18] := 1.0;
   DATA[576,19] := 2.0;
   DATA[576,20] := 148.808;
   DATA[576,21] := 155.678;
   DATA[576,22] := 1.717746;
   DATA[576,23] := 989.5155;
   DATA[576,24] := 2.0;
   DATA[576,25] := 2.0;
   DATA[576,26] := 7.880544;
   DATA[576,27] := 144.9116;
   DATA[576,28] := 263.4261;
   DATA[576,29] := 12.07383;
   DATA[576,30] := 1.728531;
   DATA[576,31] := 1.291405;
   DATA[576,32] := 0.7355248;
   DATA[576,33] := 0.3083624;
   DATA[576,34] := 2.0;
   DATA[576,35] := 250.9933;
   DATA[576,36] := 1.665972;
   DATA[576,37] := 189.743;
   DATA[576,38] := 0.000128152;
   DATA[576,39] := 1.0;
   DATA[577,0] := 2.428979;
   DATA[577,1] := 532.6992;
   DATA[577,2] := 2.0;
   DATA[577,3] := 2.0;
   DATA[577,4] := 262.1764;
   DATA[577,5] := 8.394835;
   DATA[577,6] := 327.839;
   DATA[577,7] := 2.442188;
   DATA[577,8] := 2.0;
   DATA[577,9] := 2.0;
   DATA[577,10] := 2.0;
   DATA[577,11] := 19.74838;
   DATA[577,12] := 2.209525;
   DATA[577,13] := 980.7582;
   DATA[577,14] := 1.0;
   DATA[577,15] := 2.0;
   DATA[577,16] := 1.0;
   DATA[577,17] := 1.0;
   DATA[577,18] := 1.0;
   DATA[577,19] := 2.0;
   DATA[577,20] := 148.808;
   DATA[577,21] := 155.678;
   DATA[577,22] := 1.717746;
   DATA[577,23] := 989.7847;
   DATA[577,24] := 2.0;
   DATA[577,25] := 2.0;
   DATA[577,26] := 7.880544;
   DATA[577,27] := 144.9116;
   DATA[577,28] := 263.3299;
   DATA[577,29] := 12.07383;
   DATA[577,30] := 1.728531;
   DATA[577,31] := 1.280902;
   DATA[577,32] := 0.7355248;
   DATA[577,33] := 0.3083624;
   DATA[577,34] := 2.0;
   DATA[577,35] := 250.9933;
   DATA[577,36] := 1.665972;
   DATA[577,37] := 189.743;
   DATA[577,38] := 0.000128152;
   DATA[577,39] := 1.0;
   DATA[578,0] := 2.458444;
   DATA[578,1] := 532.7384;
   DATA[578,2] := 2.0;
   DATA[578,3] := 2.0;
   DATA[578,4] := 262.1764;
   DATA[578,5] := 8.394835;
   DATA[578,6] := 327.839;
   DATA[578,7] := 2.44411;
   DATA[578,8] := 2.0;
   DATA[578,9] := 2.0;
   DATA[578,10] := 2.0;
   DATA[578,11] := 19.74838;
   DATA[578,12] := 2.207475;
   DATA[578,13] := 980.8383;
   DATA[578,14] := 1.0;
   DATA[578,15] := 2.0;
   DATA[578,16] := 1.0;
   DATA[578,17] := 1.0;
   DATA[578,18] := 1.0;
   DATA[578,19] := 2.0;
   DATA[578,20] := 148.808;
   DATA[578,21] := 155.678;
   DATA[578,22] := 1.717746;
   DATA[578,23] := 989.8616;
   DATA[578,24] := 2.0;
   DATA[578,25] := 2.0;
   DATA[578,26] := 7.880544;
   DATA[578,27] := 144.9116;
   DATA[578,28] := 263.3299;
   DATA[578,29] := 12.07383;
   DATA[578,30] := 1.728531;
   DATA[578,31] := 1.263097;
   DATA[578,32] := 0.7355248;
   DATA[578,33] := 0.3083624;
   DATA[578,34] := 2.0;
   DATA[578,35] := 250.9933;
   DATA[578,36] := 1.665972;
   DATA[578,37] := 189.743;
   DATA[578,38] := 0.000128152;
   DATA[578,39] := 1.0;
   DATA[579,0] := 2.495596;
   DATA[579,1] := 533.3272;
   DATA[579,2] := 2.0;
   DATA[579,3] := 2.0;
   DATA[579,4] := 262.1764;
   DATA[579,5] := 8.394835;
   DATA[579,6] := 327.839;
   DATA[579,7] := 2.442956;
   DATA[579,8] := 2.0;
   DATA[579,9] := 2.0;
   DATA[579,10] := 2.0;
   DATA[579,11] := 19.74838;
   DATA[579,12] := 2.206066;
   DATA[579,13] := 981.0786;
   DATA[579,14] := 1.0;
   DATA[579,15] := 2.0;
   DATA[579,16] := 1.0;
   DATA[579,17] := 1.0;
   DATA[579,18] := 1.0;
   DATA[579,19] := 2.0;
   DATA[579,20] := 148.808;
   DATA[579,21] := 155.678;
   DATA[579,22] := 1.715952;
   DATA[579,23] := 989.7847;
   DATA[579,24] := 2.0;
   DATA[579,25] := 2.0;
   DATA[579,26] := 7.880544;
   DATA[579,27] := 144.9116;
   DATA[579,28] := 263.3299;
   DATA[579,29] := 12.07383;
   DATA[579,30] := 1.728531;
   DATA[579,31] := 1.261816;
   DATA[579,32] := 0.7355248;
   DATA[579,33] := 0.3083624;
   DATA[579,34] := 2.0;
   DATA[579,35] := 250.9933;
   DATA[579,36] := 1.778105;
   DATA[579,37] := 189.743;
   DATA[579,38] := 0.000128152;
   DATA[579,39] := 1.0;
   DATA[580,0] := 2.535311;
   DATA[580,1] := 533.5235;
   DATA[580,2] := 2.0;
   DATA[580,3] := 2.0;
   DATA[580,4] := 262.1764;
   DATA[580,5] := 8.394835;
   DATA[580,6] := 327.9672;
   DATA[580,7] := 2.440906;
   DATA[580,8] := 2.0;
   DATA[580,9] := 2.0;
   DATA[580,10] := 2.0;
   DATA[580,11] := 19.74838;
   DATA[580,12] := 2.208884;
   DATA[580,13] := 981.2388;
   DATA[580,14] := 1.0;
   DATA[580,15] := 2.0;
   DATA[580,16] := 1.0;
   DATA[580,17] := 1.0;
   DATA[580,18] := 1.0;
   DATA[580,19] := 2.0;
   DATA[580,20] := 148.808;
   DATA[580,21] := 155.678;
   DATA[580,22] := 1.715952;
   DATA[580,23] := 990.4384;
   DATA[580,24] := 2.0;
   DATA[580,25] := 2.0;
   DATA[580,26] := 7.880544;
   DATA[580,27] := 145.0397;
   DATA[580,28] := 263.3299;
   DATA[580,29] := 12.07383;
   DATA[580,30] := 1.728531;
   DATA[580,31] := 1.270911;
   DATA[580,32] := 0.7355248;
   DATA[580,33] := 0.3083624;
   DATA[580,34] := 2.0;
   DATA[580,35] := 250.8011;
   DATA[580,36] := 1.778105;
   DATA[580,37] := 189.6789;
   DATA[580,38] := 0.000128152;
   DATA[580,39] := 1.0;
   DATA[581,0] := 2.571182;
   DATA[581,1] := 533.4843;
   DATA[581,2] := 2.0;
   DATA[581,3] := 2.0;
   DATA[581,4] := 262.1764;
   DATA[581,5] := 8.394835;
   DATA[581,6] := 327.9672;
   DATA[581,7] := 2.438984;
   DATA[581,8] := 2.0;
   DATA[581,9] := 2.0;
   DATA[581,10] := 2.0;
   DATA[581,11] := 19.85082;
   DATA[581,12] := 2.208884;
   DATA[581,13] := 981.2789;
   DATA[581,14] := 1.0;
   DATA[581,15] := 2.0;
   DATA[581,16] := 1.0;
   DATA[581,17] := 1.0;
   DATA[581,18] := 1.0;
   DATA[581,19] := 2.0;
   DATA[581,20] := 148.808;
   DATA[581,21] := 155.678;
   DATA[581,22] := 1.713389;
   DATA[581,23] := 990.2461;
   DATA[581,24] := 2.0;
   DATA[581,25] := 2.0;
   DATA[581,26] := 7.880544;
   DATA[581,27] := 145.0397;
   DATA[581,28] := 263.3299;
   DATA[581,29] := 12.07383;
   DATA[581,30] := 1.728531;
   DATA[581,31] := 1.288587;
   DATA[581,32] := 0.7355248;
   DATA[581,33] := 0.3083624;
   DATA[581,34] := 2.0;
   DATA[581,35] := 250.8011;
   DATA[581,36] := 1.778105;
   DATA[581,37] := 189.6148;
   DATA[581,38] := 0.000128152;
   DATA[581,39] := 1.0;
   DATA[582,0] := 2.571182;
   DATA[582,1] := 533.4843;
   DATA[582,2] := 2.0;
   DATA[582,3] := 2.0;
   DATA[582,4] := 262.1764;
   DATA[582,5] := 8.394835;
   DATA[582,6] := 327.9672;
   DATA[582,7] := 2.438984;
   DATA[582,8] := 2.0;
   DATA[582,9] := 2.0;
   DATA[582,10] := 2.0;
   DATA[582,11] := 19.85082;
   DATA[582,12] := 2.208884;
   DATA[582,13] := 981.2789;
   DATA[582,14] := 1.0;
   DATA[582,15] := 2.0;
   DATA[582,16] := 1.0;
   DATA[582,17] := 1.0;
   DATA[582,18] := 1.0;
   DATA[582,19] := 2.0;
   DATA[582,20] := 148.808;
   DATA[582,21] := 155.678;
   DATA[582,22] := 1.713389;
   DATA[582,23] := 990.2461;
   DATA[582,24] := 2.0;
   DATA[582,25] := 2.0;
   DATA[582,26] := 7.880544;
   DATA[582,27] := 145.0397;
   DATA[582,28] := 263.3299;
   DATA[582,29] := 12.07383;
   DATA[582,30] := 1.728531;
   DATA[582,31] := 1.288587;
   DATA[582,32] := 0.7355248;
   DATA[582,33] := 0.3083624;
   DATA[582,34] := 2.0;
   DATA[582,35] := 250.8011;
   DATA[582,36] := 1.778105;
   DATA[582,37] := 189.6148;
   DATA[582,38] := 0.000128152;
   DATA[582,39] := 1.0;
   DATA[583,0] := 2.60417;
   DATA[583,1] := 533.131;
   DATA[583,2] := 2.0;
   DATA[583,3] := 2.0;
   DATA[583,4] := 262.1764;
   DATA[583,5] := 8.394835;
   DATA[583,6] := 327.9672;
   DATA[583,7] := 2.438984;
   DATA[583,8] := 2.0;
   DATA[583,9] := 2.0;
   DATA[583,10] := 2.0;
   DATA[583,11] := 19.85082;
   DATA[583,12] := 2.208884;
   DATA[583,13] := 981.0786;
   DATA[583,14] := 1.0;
   DATA[583,15] := 2.0;
   DATA[583,16] := 1.0;
   DATA[583,17] := 1.0;
   DATA[583,18] := 1.0;
   DATA[583,19] := 2.0;
   DATA[583,20] := 148.808;
   DATA[583,21] := 155.678;
   DATA[583,22] := 1.713261;
   DATA[583,23] := 990.0154;
   DATA[583,24] := 2.0;
   DATA[583,25] := 2.0;
   DATA[583,26] := 7.880544;
   DATA[583,27] := 145.0397;
   DATA[583,28] := 263.3299;
   DATA[583,29] := 12.07383;
   DATA[583,30] := 1.728531;
   DATA[583,31] := 1.300372;
   DATA[583,32] := 0.7355248;
   DATA[583,33] := 0.3083624;
   DATA[583,34] := 2.0;
   DATA[583,35] := 250.8011;
   DATA[583,36] := 1.649953;
   DATA[583,37] := 189.6148;
   DATA[583,38] := 0.000128152;
   DATA[583,39] := 1.0;
   DATA[584,0] := 2.628831;
   DATA[584,1] := 533.3272;
   DATA[584,2] := 2.0;
   DATA[584,3] := 2.0;
   DATA[584,4] := 262.1764;
   DATA[584,5] := 8.394835;
   DATA[584,6] := 327.9672;
   DATA[584,7] := 2.438984;
   DATA[584,8] := 2.0;
   DATA[584,9] := 2.0;
   DATA[584,10] := 2.0;
   DATA[584,11] := 19.85082;
   DATA[584,12] := 2.208884;
   DATA[584,13] := 981.7595;
   DATA[584,14] := 1.0;
   DATA[584,15] := 2.0;
   DATA[584,16] := 1.0;
   DATA[584,17] := 1.0;
   DATA[584,18] := 1.0;
   DATA[584,19] := 2.0;
   DATA[584,20] := 148.808;
   DATA[584,21] := 155.678;
   DATA[584,22] := 1.713261;
   DATA[584,23] := 990.0923;
   DATA[584,24] := 2.0;
   DATA[584,25] := 2.0;
   DATA[584,26] := 7.880544;
   DATA[584,27] := 145.0397;
   DATA[584,28] := 263.3299;
   DATA[584,29] := 12.15073;
   DATA[584,30] := 1.726609;
   DATA[584,31] := 1.30114;
   DATA[584,32] := 0.7355248;
   DATA[584,33] := 0.3083624;
   DATA[584,34] := 2.0;
   DATA[584,35] := 250.8011;
   DATA[584,36] := 1.649953;
   DATA[584,37] := 189.6148;
   DATA[584,38] := 0.000128152;
   DATA[584,39] := 1.0;
   DATA[585,0] := 2.647407;
   DATA[585,1] := 533.445;
   DATA[585,2] := 2.0;
   DATA[585,3] := 2.0;
   DATA[585,4] := 262.1764;
   DATA[585,5] := 8.394835;
   DATA[585,6] := 327.9672;
   DATA[585,7] := 2.440137;
   DATA[585,8] := 2.0;
   DATA[585,9] := 2.0;
   DATA[585,10] := 2.0;
   DATA[585,11] := 19.85082;
   DATA[585,12] := 2.208884;
   DATA[585,13] := 981.8396;
   DATA[585,14] := 1.0;
   DATA[585,15] := 2.0;
   DATA[585,16] := 1.0;
   DATA[585,17] := 1.0;
   DATA[585,18] := 1.0;
   DATA[585,19] := 2.0;
   DATA[585,20] := 148.808;
   DATA[585,21] := 155.678;
   DATA[585,22] := 1.712363;
   DATA[585,23] := 990.0154;
   DATA[585,24] := 2.0;
   DATA[585,25] := 2.0;
   DATA[585,26] := 7.880544;
   DATA[585,27] := 145.0397;
   DATA[585,28] := 263.3299;
   DATA[585,29] := 12.15073;
   DATA[585,30] := 1.724814;
   DATA[585,31] := 1.30114;
   DATA[585,32] := 0.7355248;
   DATA[585,33] := 0.3083624;
   DATA[585,34] := 2.0;
   DATA[585,35] := 250.6729;
   DATA[585,36] := 1.649953;
   DATA[585,37] := 189.5187;
   DATA[585,38] := 0.000128152;
   DATA[585,39] := 1.0;
   DATA[586,0] := 2.64997;
   DATA[586,1] := 533.1702;
   DATA[586,2] := 2.0;
   DATA[586,3] := 2.0;
   DATA[586,4] := 262.1764;
   DATA[586,5] := 8.394835;
   DATA[586,6] := 327.9672;
   DATA[586,7] := 2.440521;
   DATA[586,8] := 2.0;
   DATA[586,9] := 2.0;
   DATA[586,10] := 2.0;
   DATA[586,11] := 19.85082;
   DATA[586,12] := 2.208884;
   DATA[586,13] := 982.2802;
   DATA[586,14] := 1.0;
   DATA[586,15] := 2.0;
   DATA[586,16] := 1.0;
   DATA[586,17] := 1.0;
   DATA[586,18] := 1.0;
   DATA[586,19] := 2.0;
   DATA[586,20] := 148.808;
   DATA[586,21] := 155.678;
   DATA[586,22] := 1.712363;
   DATA[586,23] := 990.0154;
   DATA[586,24] := 2.0;
   DATA[586,25] := 2.0;
   DATA[586,26] := 7.880544;
   DATA[586,27] := 145.0397;
   DATA[586,28] := 263.3299;
   DATA[586,29] := 12.15073;
   DATA[586,30] := 1.724814;
   DATA[586,31] := 1.285513;
   DATA[586,32] := 0.7355248;
   DATA[586,33] := 0.3083624;
   DATA[586,34] := 2.0;
   DATA[586,35] := 250.5127;
   DATA[586,36] := 1.649953;
   DATA[586,37] := 189.3745;
   DATA[586,38] := 0.000128152;
   DATA[586,39] := 1.0;
   DATA[587,0] := 2.632034;
   DATA[587,1] := 533.1702;
   DATA[587,2] := 2.0;
   DATA[587,3] := 2.0;
   DATA[587,4] := 262.1764;
   DATA[587,5] := 8.394835;
   DATA[587,6] := 327.9672;
   DATA[587,7] := 2.440521;
   DATA[587,8] := 2.0;
   DATA[587,9] := 2.0;
   DATA[587,10] := 2.0;
   DATA[587,11] := 19.8028;
   DATA[587,12] := 2.208884;
   DATA[587,13] := 982.7609;
   DATA[587,14] := 1.0;
   DATA[587,15] := 2.0;
   DATA[587,16] := 1.0;
   DATA[587,17] := 1.0;
   DATA[587,18] := 1.0;
   DATA[587,19] := 2.0;
   DATA[587,20] := 148.808;
   DATA[587,21] := 155.7037;
   DATA[587,22] := 1.712363;
   DATA[587,23] := 990.1692;
   DATA[587,24] := 2.0;
   DATA[587,25] := 2.0;
   DATA[587,26] := 7.880544;
   DATA[587,27] := 145.0397;
   DATA[587,28] := 263.3299;
   DATA[587,29] := 12.15073;
   DATA[587,30] := 1.724814;
   DATA[587,31] := 1.282823;
   DATA[587,32] := 0.7355248;
   DATA[587,33] := 0.3083624;
   DATA[587,34] := 2.0;
   DATA[587,35] := 250.5127;
   DATA[587,36] := 1.649953;
   DATA[587,37] := 189.3745;
   DATA[587,38] := 0.000128152;
   DATA[587,39] := 1.0;
   DATA[588,0] := 2.621145;
   DATA[588,1] := 533.3665;
   DATA[588,2] := 2.0;
   DATA[588,3] := 2.0;
   DATA[588,4] := 262.1764;
   DATA[588,5] := 8.394835;
   DATA[588,6] := 327.9672;
   DATA[588,7] := 2.440521;
   DATA[588,8] := 2.0;
   DATA[588,9] := 2.0;
   DATA[588,10] := 2.0;
   DATA[588,11] := 19.8028;
   DATA[588,12] := 2.208884;
   DATA[588,13] := 983.1614;
   DATA[588,14] := 1.0;
   DATA[588,15] := 2.0;
   DATA[588,16] := 1.0;
   DATA[588,17] := 1.0;
   DATA[588,18] := 1.0;
   DATA[588,19] := 2.0;
   DATA[588,20] := 148.808;
   DATA[588,21] := 155.7293;
   DATA[588,22] := 1.714542;
   DATA[588,23] := 990.3615;
   DATA[588,24] := 2.0;
   DATA[588,25] := 2.0;
   DATA[588,26] := 7.880544;
   DATA[588,27] := 145.0397;
   DATA[588,28] := 263.3299;
   DATA[588,29] := 12.15073;
   DATA[588,30] := 1.724814;
   DATA[588,31] := 1.287691;
   DATA[588,32] := 0.7355248;
   DATA[588,33] := 0.3083624;
   DATA[588,34] := 2.0;
   DATA[588,35] := 250.5127;
   DATA[588,36] := 1.649953;
   DATA[588,37] := 189.3745;
   DATA[588,38] := 0.000128152;
   DATA[588,39] := 1.0;
   DATA[589,0] := 2.613138;
   DATA[589,1] := 533.0917;
   DATA[589,2] := 2.0;
   DATA[589,3] := 2.0;
   DATA[589,4] := 262.1764;
   DATA[589,5] := 8.394835;
   DATA[589,6] := 327.9672;
   DATA[589,7] := 2.440521;
   DATA[589,8] := 2.0;
   DATA[589,9] := 2.0;
   DATA[589,10] := 2.0;
   DATA[589,11] := 19.84442;
   DATA[589,12] := 2.208884;
   DATA[589,13] := 983.4818;
   DATA[589,14] := 1.0;
   DATA[589,15] := 2.0;
   DATA[589,16] := 1.0;
   DATA[589,17] := 1.0;
   DATA[589,18] := 1.0;
   DATA[589,19] := 2.0;
   DATA[589,20] := 148.808;
   DATA[589,21] := 155.7293;
   DATA[589,22] := 1.714542;
   DATA[589,23] := 990.4768;
   DATA[589,24] := 2.0;
   DATA[589,25] := 2.0;
   DATA[589,26] := 7.880544;
   DATA[589,27] := 145.0397;
   DATA[589,28] := 263.3299;
   DATA[589,29] := 12.15073;
   DATA[589,30] := 1.724814;
   DATA[589,31] := 1.282951;
   DATA[589,32] := 0.7355248;
   DATA[589,33] := 0.3083624;
   DATA[589,34] := 2.0;
   DATA[589,35] := 250.5127;
   DATA[589,36] := 1.649953;
   DATA[589,37] := 189.3745;
   DATA[589,38] := 0.000128152;
   DATA[589,39] := 1.0;
   DATA[590,0] := 2.605131;
   DATA[590,1] := 533.0524;
   DATA[590,2] := 2.0;
   DATA[590,3] := 2.0;
   DATA[590,4] := 262.1764;
   DATA[590,5] := 8.394835;
   DATA[590,6] := 327.9672;
   DATA[590,7] := 2.441162;
   DATA[590,8] := 2.0;
   DATA[590,9] := 2.0;
   DATA[590,10] := 2.0;
   DATA[590,11] := 19.84442;
   DATA[590,12] := 2.208884;
   DATA[590,13] := 983.8423;
   DATA[590,14] := 1.0;
   DATA[590,15] := 2.0;
   DATA[590,16] := 1.0;
   DATA[590,17] := 1.0;
   DATA[590,18] := 1.0;
   DATA[590,19] := 2.0;
   DATA[590,20] := 148.808;
   DATA[590,21] := 155.7293;
   DATA[590,22] := 1.714542;
   DATA[590,23] := 990.2845;
   DATA[590,24] := 2.0;
   DATA[590,25] := 2.0;
   DATA[590,26] := 7.880544;
   DATA[590,27] := 145.0397;
   DATA[590,28] := 263.3299;
   DATA[590,29] := 12.15073;
   DATA[590,30] := 1.724814;
   DATA[590,31] := 1.27296;
   DATA[590,32] := 0.7355248;
   DATA[590,33] := 0.3083624;
   DATA[590,34] := 2.0;
   DATA[590,35] := 250.5127;
   DATA[590,36] := 1.649953;
   DATA[590,37] := 189.3745;
   DATA[590,38] := 0.000128152;
   DATA[590,39] := 1.0;
   DATA[591,0] := 2.588156;
   DATA[591,1] := 532.8954;
   DATA[591,2] := 2.0;
   DATA[591,3] := 2.0;
   DATA[591,4] := 262.1764;
   DATA[591,5] := 8.394835;
   DATA[591,6] := 327.6596;
   DATA[591,7] := 2.441162;
   DATA[591,8] := 2.0;
   DATA[591,9] := 2.0;
   DATA[591,10] := 2.0;
   DATA[591,11] := 19.77399;
   DATA[591,12] := 2.208884;
   DATA[591,13] := 984.4031;
   DATA[591,14] := 1.0;
   DATA[591,15] := 2.0;
   DATA[591,16] := 1.0;
   DATA[591,17] := 1.0;
   DATA[591,18] := 1.0;
   DATA[591,19] := 2.0;
   DATA[591,20] := 148.808;
   DATA[591,21] := 155.7293;
   DATA[591,22] := 1.714542;
   DATA[591,23] := 990.5537;
   DATA[591,24] := 2.0;
   DATA[591,25] := 2.0;
   DATA[591,26] := 7.880544;
   DATA[591,27] := 145.0397;
   DATA[591,28] := 263.3299;
   DATA[591,29] := 12.15073;
   DATA[591,30] := 1.724045;
   DATA[591,31] := 1.271423;
   DATA[591,32] := 0.7355248;
   DATA[591,33] := 0.3083624;
   DATA[591,34] := 2.0;
   DATA[591,35] := 250.5127;
   DATA[591,36] := 1.649953;
   DATA[591,37] := 189.3745;
   DATA[591,38] := 0.000128152;
   DATA[591,39] := 1.0;
   DATA[592,0] := 2.56958;
   DATA[592,1] := 532.6599;
   DATA[592,2] := 2.0;
   DATA[592,3] := 2.0;
   DATA[592,4] := 262.1764;
   DATA[592,5] := 8.394835;
   DATA[592,6] := 327.6596;
   DATA[592,7] := 2.441162;
   DATA[592,8] := 2.0;
   DATA[592,9] := 2.0;
   DATA[592,10] := 2.0;
   DATA[592,11] := 19.72598;
   DATA[592,12] := 2.208884;
   DATA[592,13] := 985.0038;
   DATA[592,14] := 1.0;
   DATA[592,15] := 2.0;
   DATA[592,16] := 1.0;
   DATA[592,17] := 1.0;
   DATA[592,18] := 1.0;
   DATA[592,19] := 2.0;
   DATA[592,20] := 148.808;
   DATA[592,21] := 155.7293;
   DATA[592,22] := 1.715439;
   DATA[592,23] := 990.3999;
   DATA[592,24] := 2.0;
   DATA[592,25] := 2.0;
   DATA[592,26] := 7.880544;
   DATA[592,27] := 145.0397;
   DATA[592,28] := 263.3299;
   DATA[592,29] := 12.15073;
   DATA[592,30] := 1.724045;
   DATA[592,31] := 1.273345;
   DATA[592,32] := 0.7355248;
   DATA[592,33] := 0.3083624;
   DATA[592,34] := 2.0;
   DATA[592,35] := 250.5127;
   DATA[592,36] := 1.649953;
   DATA[592,37] := 189.3745;
   DATA[592,38] := 0.000128152;
   DATA[592,39] := 1.0;
   DATA[593,0] := 2.556129;
   DATA[593,1] := 532.3851;
   DATA[593,2] := 2.0;
   DATA[593,3] := 2.0;
   DATA[593,4] := 262.1764;
   DATA[593,5] := 8.396116;
   DATA[593,6] := 327.6596;
   DATA[593,7] := 2.439753;
   DATA[593,8] := 2.0;
   DATA[593,9] := 2.0;
   DATA[593,10] := 2.0;
   DATA[593,11] := 19.72598;
   DATA[593,12] := 2.208884;
   DATA[593,13] := 985.1641;
   DATA[593,14] := 1.0;
   DATA[593,15] := 2.0;
   DATA[593,16] := 1.0;
   DATA[593,17] := 1.0;
   DATA[593,18] := 1.0;
   DATA[593,19] := 2.0;
   DATA[593,20] := 148.808;
   DATA[593,21] := 155.7293;
   DATA[593,22] := 1.715439;
   DATA[593,23] := 990.746;
   DATA[593,24] := 2.0;
   DATA[593,25] := 2.0;
   DATA[593,26] := 7.880544;
   DATA[593,27] := 145.0397;
   DATA[593,28] := 263.1377;
   DATA[593,29] := 12.15073;
   DATA[593,30] := 1.724045;
   DATA[593,31] := 1.277699;
   DATA[593,32] := 0.7355248;
   DATA[593,33] := 0.3083624;
   DATA[593,34] := 2.0;
   DATA[593,35] := 250.5127;
   DATA[593,36] := 1.649953;
   DATA[593,37] := 189.3745;
   DATA[593,38] := 0.000128152;
   DATA[593,39] := 1.0;
   DATA[594,0] := 2.542677;
   DATA[594,1] := 532.1104;
   DATA[594,2] := 2.0;
   DATA[594,3] := 2.0;
   DATA[594,4] := 262.1764;
   DATA[594,5] := 8.396116;
   DATA[594,6] := 327.6596;
   DATA[594,7] := 2.439753;
   DATA[594,8] := 2.0;
   DATA[594,9] := 2.0;
   DATA[594,10] := 2.0;
   DATA[594,11] := 19.66195;
   DATA[594,12] := 2.208884;
   DATA[594,13] := 985.6848;
   DATA[594,14] := 1.0;
   DATA[594,15] := 2.0;
   DATA[594,16] := 1.0;
   DATA[594,17] := 1.0;
   DATA[594,18] := 1.0;
   DATA[594,19] := 2.0;
   DATA[594,20] := 148.808;
   DATA[594,21] := 155.7293;
   DATA[594,22] := 1.717105;
   DATA[594,23] := 990.4384;
   DATA[594,24] := 2.0;
   DATA[594,25] := 2.0;
   DATA[594,26] := 7.880544;
   DATA[594,27] := 145.0397;
   DATA[594,28] := 263.1377;
   DATA[594,29] := 12.15073;
   DATA[594,30] := 1.726352;
   DATA[594,31] := 1.272576;
   DATA[594,32] := 0.7355248;
   DATA[594,33] := 0.3083624;
   DATA[594,34] := 2.0;
   DATA[594,35] := 250.5928;
   DATA[594,36] := 1.649953;
   DATA[594,37] := 189.3745;
   DATA[594,38] := 0.000128152;
   DATA[594,39] := 1.0;
   DATA[595,0] := 2.521218;
   DATA[595,1] := 532.1104;
   DATA[595,2] := 2.0;
   DATA[595,3] := 2.0;
   DATA[595,4] := 262.1764;
   DATA[595,5] := 8.396116;
   DATA[595,6] := 327.8647;
   DATA[595,7] := 2.439753;
   DATA[595,8] := 2.0;
   DATA[595,9] := 2.0;
   DATA[595,10] := 2.0;
   DATA[595,11] := 19.65555;
   DATA[595,12] := 2.209013;
   DATA[595,13] := 986.2055;
   DATA[595,14] := 1.0;
   DATA[595,15] := 2.0;
   DATA[595,16] := 1.0;
   DATA[595,17] := 1.0;
   DATA[595,18] := 1.0;
   DATA[595,19] := 2.0;
   DATA[595,20] := 148.808;
   DATA[595,21] := 155.7293;
   DATA[595,22] := 1.717361;
   DATA[595,23] := 990.4384;
   DATA[595,24] := 2.0;
   DATA[595,25] := 2.0;
   DATA[595,26] := 7.880544;
   DATA[595,27] := 145.0397;
   DATA[595,28] := 263.1377;
   DATA[595,29] := 12.15073;
   DATA[595,30] := 1.726993;
   DATA[595,31] := 1.25823;
   DATA[595,32] := 0.7355248;
   DATA[595,33] := 0.3083624;
   DATA[595,34] := 2.0;
   DATA[595,35] := 250.753;
   DATA[595,36] := 1.649953;
   DATA[595,37] := 189.3745;
   DATA[595,38] := 0.000128152;
   DATA[595,39] := 1.0;
   DATA[596,0] := 2.508728;
   DATA[596,1] := 531.6001;
   DATA[596,2] := 2.0;
   DATA[596,3] := 2.0;
   DATA[596,4] := 262.1764;
   DATA[596,5] := 8.396116;
   DATA[596,6] := 327.8647;
   DATA[596,7] := 2.442188;
   DATA[596,8] := 2.0;
   DATA[596,9] := 2.0;
   DATA[596,10] := 2.0;
   DATA[596,11] := 19.65555;
   DATA[596,12] := 2.209909;
   DATA[596,13] := 986.1654;
   DATA[596,14] := 1.0;
   DATA[596,15] := 2.0;
   DATA[596,16] := 1.0;
   DATA[596,17] := 1.0;
   DATA[596,18] := 1.0;
   DATA[596,19] := 2.0;
   DATA[596,20] := 148.808;
   DATA[596,21] := 155.7293;
   DATA[596,22] := 1.717361;
   DATA[596,23] := 990.6306;
   DATA[596,24] := 2.0;
   DATA[596,25] := 2.0;
   DATA[596,26] := 7.880544;
   DATA[596,27] := 145.0397;
   DATA[596,28] := 263.1377;
   DATA[596,29] := 12.15073;
   DATA[596,30] := 1.726993;
   DATA[596,31] := 1.254515;
   DATA[596,32] := 0.7355248;
   DATA[596,33] := 0.3083624;
   DATA[596,34] := 2.0;
   DATA[596,35] := 250.753;
   DATA[596,36] := 1.649953;
   DATA[596,37] := 189.4066;
   DATA[596,38] := 0.000128152;
   DATA[596,39] := 1.0;
   DATA[597,0] := 2.48823;
   DATA[597,1] := 531.9534;
   DATA[597,2] := 2.0;
   DATA[597,3] := 2.0;
   DATA[597,4] := 262.1764;
   DATA[597,5] := 8.396116;
   DATA[597,6] := 327.8647;
   DATA[597,7] := 2.442188;
   DATA[597,8] := 2.0;
   DATA[597,9] := 2.0;
   DATA[597,10] := 2.0;
   DATA[597,11] := 19.65555;
   DATA[597,12] := 2.212343;
   DATA[597,13] := 986.0853;
   DATA[597,14] := 1.0;
   DATA[597,15] := 2.0;
   DATA[597,16] := 1.0;
   DATA[597,17] := 1.0;
   DATA[597,18] := 1.0;
   DATA[597,19] := 2.0;
   DATA[597,20] := 148.808;
   DATA[597,21] := 155.7293;
   DATA[597,22] := 1.717361;
   DATA[597,23] := 990.5922;
   DATA[597,24] := 2.0;
   DATA[597,25] := 2.0;
   DATA[597,26] := 7.880544;
   DATA[597,27] := 145.0397;
   DATA[597,28] := 263.1377;
   DATA[597,29] := 12.15073;
   DATA[597,30] := 1.726993;
   DATA[597,31] := 1.258102;
   DATA[597,32] := 0.7355248;
   DATA[597,33] := 0.3083624;
   DATA[597,34] := 2.0;
   DATA[597,35] := 250.8171;
   DATA[597,36] := 1.649953;
   DATA[597,37] := 189.6629;
   DATA[597,38] := 0.000128152;
   DATA[597,39] := 1.0;
   DATA[598,0] := 2.47702;
   DATA[598,1] := 532.3066;
   DATA[598,2] := 2.0;
   DATA[598,3] := 2.0;
   DATA[598,4] := 262.1764;
   DATA[598,5] := 8.396116;
   DATA[598,6] := 327.8647;
   DATA[598,7] := 2.440137;
   DATA[598,8] := 2.0;
   DATA[598,9] := 2.0;
   DATA[598,10] := 2.0;
   DATA[598,11] := 19.70677;
   DATA[598,12] := 2.212343;
   DATA[598,13] := 986.0052;
   DATA[598,14] := 1.0;
   DATA[598,15] := 2.0;
   DATA[598,16] := 1.0;
   DATA[598,17] := 1.0;
   DATA[598,18] := 1.0;
   DATA[598,19] := 2.0;
   DATA[598,20] := 148.808;
   DATA[598,21] := 155.7806;
   DATA[598,22] := 1.718387;
   DATA[598,23] := 990.8229;
   DATA[598,24] := 2.0;
   DATA[598,25] := 2.0;
   DATA[598,26] := 7.880544;
   DATA[598,27] := 145.0397;
   DATA[598,28] := 263.1377;
   DATA[598,29] := 12.15073;
   DATA[598,30] := 1.726993;
   DATA[598,31] := 1.278468;
   DATA[598,32] := 0.7355248;
   DATA[598,33] := 0.3083624;
   DATA[598,34] := 2.0;
   DATA[598,35] := 250.8972;
   DATA[598,36] := 1.649953;
   DATA[598,37] := 189.6789;
   DATA[598,38] := 0.000128152;
   DATA[598,39] := 1.0;
   DATA[599,0] := 2.460045;
   DATA[599,1] := 533.1702;
   DATA[599,2] := 2.0;
   DATA[599,3] := 2.0;
   DATA[599,4] := 262.1764;
   DATA[599,5] := 8.396116;
   DATA[599,6] := 327.8647;
   DATA[599,7] := 2.439625;
   DATA[599,8] := 2.0;
   DATA[599,9] := 2.0;
   DATA[599,10] := 2.0;
   DATA[599,11] := 19.71637;
   DATA[599,12] := 2.212343;
   DATA[599,13] := 986.3657;
   DATA[599,14] := 1.0;
   DATA[599,15] := 2.0;
   DATA[599,16] := 1.0;
   DATA[599,17] := 1.0;
   DATA[599,18] := 1.0;
   DATA[599,19] := 2.0;
   DATA[599,20] := 148.808;
   DATA[599,21] := 155.7806;
   DATA[599,22] := 1.719156;
   DATA[599,23] := 990.9382;
   DATA[599,24] := 2.0;
   DATA[599,25] := 2.0;
   DATA[599,26] := 7.880544;
   DATA[599,27] := 145.0397;
   DATA[599,28] := 263.1377;
   DATA[599,29] := 12.15073;
   DATA[599,30] := 1.728019;
   DATA[599,31] := 1.297682;
   DATA[599,32] := 0.7355248;
   DATA[599,33] := 0.3083624;
   DATA[599,34] := 2.0;
   DATA[599,35] := 250.8972;
   DATA[599,36] := 1.649953;
   DATA[599,37] := 189.6789;
   DATA[599,38] := 0.000128152;
   DATA[599,39] := 1.0;
   DATA[600,0] := 2.446594;
   DATA[600,1] := 533.759;
   DATA[600,2] := 2.0;
   DATA[600,3] := 2.0;
   DATA[600,4] := 262.1764;
   DATA[600,5] := 8.396116;
   DATA[600,6] := 327.8647;
   DATA[600,7] := 2.439625;
   DATA[600,8] := 2.0;
   DATA[600,9] := 2.0;
   DATA[600,10] := 2.0;
   DATA[600,11] := 19.67155;
   DATA[600,12] := 2.212343;
   DATA[600,13] := 986.6461;
   DATA[600,14] := 1.0;
   DATA[600,15] := 2.0;
   DATA[600,16] := 1.0;
   DATA[600,17] := 1.0;
   DATA[600,18] := 1.0;
   DATA[600,19] := 2.0;
   DATA[600,20] := 148.808;
   DATA[600,21] := 155.7806;
   DATA[600,22] := 1.720565;
   DATA[600,23] := 990.9382;
   DATA[600,24] := 2.0;
   DATA[600,25] := 2.0;
   DATA[600,26] := 7.880544;
   DATA[600,27] := 145.0397;
   DATA[600,28] := 263.1377;
   DATA[600,29] := 12.15073;
   DATA[600,30] := 1.728659;
   DATA[600,31] := 1.297169;
   DATA[600,32] := 0.7355248;
   DATA[600,33] := 0.3075937;
   DATA[600,34] := 2.0;
   DATA[600,35] := 250.8972;
   DATA[600,36] := 1.649953;
   DATA[600,37] := 189.6789;
   DATA[600,38] := 0.000128152;
   DATA[600,39] := 1.0;
   DATA[601,0] := 2.433783;
   DATA[601,1] := 534.3085;
   DATA[601,2] := 2.0;
   DATA[601,3] := 2.0;
   DATA[601,4] := 262.1764;
   DATA[601,5] := 8.396116;
   DATA[601,6] := 327.8647;
   DATA[601,7] := 2.439625;
   DATA[601,8] := 2.0;
   DATA[601,9] := 2.0;
   DATA[601,10] := 2.0;
   DATA[601,11] := 19.67155;
   DATA[601,12] := 2.212343;
   DATA[601,13] := 987.0065;
   DATA[601,14] := 1.0;
   DATA[601,15] := 2.0;
   DATA[601,16] := 1.0;
   DATA[601,17] := 1.0;
   DATA[601,18] := 1.0;
   DATA[601,19] := 2.0;
   DATA[601,20] := 148.808;
   DATA[601,21] := 155.7806;
   DATA[601,22] := 1.720565;
   DATA[601,23] := 990.7844;
   DATA[601,24] := 2.0;
   DATA[601,25] := 2.0;
   DATA[601,26] := 7.880544;
   DATA[601,27] := 145.0397;
   DATA[601,28] := 263.1377;
   DATA[601,29] := 12.15073;
   DATA[601,30] := 1.728659;
   DATA[601,31] := 1.282823;
   DATA[601,32] := 0.7355248;
   DATA[601,33] := 0.3070813;
   DATA[601,34] := 2.0;
   DATA[601,35] := 250.8972;
   DATA[601,36] := 1.649953;
   DATA[601,37] := 189.6789;
   DATA[601,38] := 0.000128152;
   DATA[601,39] := 1.0;
   DATA[602,0] := 2.426737;
   DATA[602,1] := 534.5441;
   DATA[602,2] := 2.0;
   DATA[602,3] := 2.0;
   DATA[602,4] := 262.1764;
   DATA[602,5] := 8.396116;
   DATA[602,6] := 327.8647;
   DATA[602,7] := 2.439625;
   DATA[602,8] := 2.0;
   DATA[602,9] := 2.0;
   DATA[602,10] := 2.0;
   DATA[602,11] := 19.69396;
   DATA[602,12] := 2.212343;
   DATA[602,13] := 986.9665;
   DATA[602,14] := 1.0;
   DATA[602,15] := 2.0;
   DATA[602,16] := 1.0;
   DATA[602,17] := 1.0;
   DATA[602,18] := 1.0;
   DATA[602,19] := 2.0;
   DATA[602,20] := 148.808;
   DATA[602,21] := 155.7806;
   DATA[602,22] := 1.719156;
   DATA[602,23] := 991.0151;
   DATA[602,24] := 2.0;
   DATA[602,25] := 2.0;
   DATA[602,26] := 7.880544;
   DATA[602,27] := 145.0397;
   DATA[602,28] := 263.1377;
   DATA[602,29] := 12.15073;
   DATA[602,30] := 1.728659;
   DATA[602,31] := 1.281542;
   DATA[602,32] := 0.7355248;
   DATA[602,33] := 0.3063127;
   DATA[602,34] := 2.0;
   DATA[602,35] := 251.0254;
   DATA[602,36] := 1.649953;
   DATA[602,37] := 189.6949;
   DATA[602,38] := 0.000128152;
   DATA[602,39] := 1.0;
   DATA[603,0] := 2.426737;
   DATA[603,1] := 534.7403;
   DATA[603,2] := 2.0;
   DATA[603,3] := 2.0;
   DATA[603,4] := 262.1764;
   DATA[603,5] := 8.396116;
   DATA[603,6] := 327.8647;
   DATA[603,7] := 2.439625;
   DATA[603,8] := 2.0;
   DATA[603,9] := 2.0;
   DATA[603,10] := 2.0;
   DATA[603,11] := 19.69396;
   DATA[603,12] := 2.212343;
   DATA[603,13] := 986.6461;
   DATA[603,14] := 1.0;
   DATA[603,15] := 2.0;
   DATA[603,16] := 1.0;
   DATA[603,17] := 1.0;
   DATA[603,18] := 1.0;
   DATA[603,19] := 2.0;
   DATA[603,20] := 148.808;
   DATA[603,21] := 155.7806;
   DATA[603,22] := 1.716849;
   DATA[603,23] := 990.9382;
   DATA[603,24] := 2.0;
   DATA[603,25] := 2.0;
   DATA[603,26] := 7.880544;
   DATA[603,27] := 145.0397;
   DATA[603,28] := 263.1377;
   DATA[603,29] := 12.15073;
   DATA[603,30] := 1.728659;
   DATA[603,31] := 1.27296;
   DATA[603,32] := 0.7355248;
   DATA[603,33] := 0.3063127;
   DATA[603,34] := 2.0;
   DATA[603,35] := 251.0254;
   DATA[603,36] := 1.649953;
   DATA[603,37] := 189.759;
   DATA[603,38] := 0.000128152;
   DATA[603,39] := 1.0;
   DATA[604,0] := 2.452679;
   DATA[604,1] := 534.8973;
   DATA[604,2] := 2.0;
   DATA[604,3] := 2.0;
   DATA[604,4] := 262.1764;
   DATA[604,5] := 8.396116;
   DATA[604,6] := 327.8647;
   DATA[604,7] := 2.440137;
   DATA[604,8] := 2.0;
   DATA[604,9] := 2.0;
   DATA[604,10] := 2.0;
   DATA[604,11] := 19.69396;
   DATA[604,12] := 2.212343;
   DATA[604,13] := 986.6862;
   DATA[604,14] := 1.0;
   DATA[604,15] := 2.0;
   DATA[604,16] := 1.0;
   DATA[604,17] := 1.0;
   DATA[604,18] := 1.0;
   DATA[604,19] := 2.0;
   DATA[604,20] := 148.808;
   DATA[604,21] := 155.7806;
   DATA[604,22] := 1.716849;
   DATA[604,23] := 991.1689;
   DATA[604,24] := 2.0;
   DATA[604,25] := 2.0;
   DATA[604,26] := 7.880544;
   DATA[604,27] := 145.0397;
   DATA[604,28] := 263.1377;
   DATA[604,29] := 12.15073;
   DATA[604,30] := 1.728659;
   DATA[604,31] := 1.277443;
   DATA[604,32] := 0.7355248;
   DATA[604,33] := 0.3063127;
   DATA[604,34] := 2.0;
   DATA[604,35] := 251.0254;
   DATA[604,36] := 1.649953;
   DATA[604,37] := 189.759;
   DATA[604,38] := 0.000128152;
   DATA[604,39] := 1.0;
   DATA[605,0] := 2.503603;
   DATA[605,1] := 534.9366;
   DATA[605,2] := 2.0;
   DATA[605,3] := 2.0;
   DATA[605,4] := 262.1764;
   DATA[605,5] := 8.396116;
   DATA[605,6] := 327.8647;
   DATA[605,7] := 2.440137;
   DATA[605,8] := 2.0;
   DATA[605,9] := 2.0;
   DATA[605,10] := 2.0;
   DATA[605,11] := 19.69396;
   DATA[605,12] := 2.211575;
   DATA[605,13] := 986.7662;
   DATA[605,14] := 1.0;
   DATA[605,15] := 2.0;
   DATA[605,16] := 1.0;
   DATA[605,17] := 1.0;
   DATA[605,18] := 1.0;
   DATA[605,19] := 2.0;
   DATA[605,20] := 148.808;
   DATA[605,21] := 155.7806;
   DATA[605,22] := 1.716849;
   DATA[605,23] := 991.1305;
   DATA[605,24] := 2.0;
   DATA[605,25] := 2.0;
   DATA[605,26] := 7.880544;
   DATA[605,27] := 145.1679;
   DATA[605,28] := 263.1377;
   DATA[605,29] := 12.15073;
   DATA[605,30] := 1.728659;
   DATA[605,31] := 1.291918;
   DATA[605,32] := 0.7355248;
   DATA[605,33] := 0.3063127;
   DATA[605,34] := 2.0;
   DATA[605,35] := 251.0254;
   DATA[605,36] := 1.649953;
   DATA[605,37] := 189.759;
   DATA[605,38] := 0.000128152;
   DATA[605,39] := 1.0;
   DATA[606,0] := 2.543638;
   DATA[606,1] := 534.8581;
   DATA[606,2] := 2.0;
   DATA[606,3] := 2.0;
   DATA[606,4] := 262.1764;
   DATA[606,5] := 8.396116;
   DATA[606,6] := 327.8647;
   DATA[606,7] := 2.441675;
   DATA[606,8] := 2.0;
   DATA[606,9] := 2.0;
   DATA[606,10] := 2.0;
   DATA[606,11] := 19.74198;
   DATA[606,12] := 2.209653;
   DATA[606,13] := 986.9665;
   DATA[606,14] := 1.0;
   DATA[606,15] := 2.0;
   DATA[606,16] := 1.0;
   DATA[606,17] := 1.0;
   DATA[606,18] := 1.0;
   DATA[606,19] := 2.0;
   DATA[606,20] := 148.808;
   DATA[606,21] := 155.7806;
   DATA[606,22] := 1.71813;
   DATA[606,23] := 990.9382;
   DATA[606,24] := 2.0;
   DATA[606,25] := 2.0;
   DATA[606,26] := 7.880544;
   DATA[606,27] := 145.1679;
   DATA[606,28] := 263.1377;
   DATA[606,29] := 12.15073;
   DATA[606,30] := 1.726096;
   DATA[606,31] := 1.286282;
   DATA[606,32] := 0.7355248;
   DATA[606,33] := 0.3063127;
   DATA[606,34] := 2.0;
   DATA[606,35] := 251.0254;
   DATA[606,36] := 1.649953;
   DATA[606,37] := 189.759;
   DATA[606,38] := 0.000128152;
   DATA[606,39] := 1.0;
   DATA[607,0] := 2.579509;
   DATA[607,1] := 534.8973;
   DATA[607,2] := 2.0;
   DATA[607,3] := 2.0;
   DATA[607,4] := 262.1764;
   DATA[607,5] := 8.395475;
   DATA[607,6] := 327.8647;
   DATA[607,7] := 2.441803;
   DATA[607,8] := 2.0;
   DATA[607,9] := 2.0;
   DATA[607,10] := 2.0;
   DATA[607,11] := 19.74198;
   DATA[607,12] := 2.209653;
   DATA[607,13] := 986.566;
   DATA[607,14] := 1.0;
   DATA[607,15] := 2.0;
   DATA[607,16] := 1.0;
   DATA[607,17] := 1.0;
   DATA[607,18] := 1.0;
   DATA[607,19] := 2.0;
   DATA[607,20] := 148.808;
   DATA[607,21] := 155.7806;
   DATA[607,22] := 1.719156;
   DATA[607,23] := 991.2074;
   DATA[607,24] := 2.0;
   DATA[607,25] := 2.0;
   DATA[607,26] := 7.880544;
   DATA[607,27] := 145.1679;
   DATA[607,28] := 263.1377;
   DATA[607,29] := 12.15073;
   DATA[607,30] := 1.724173;
   DATA[607,31] := 1.287306;
   DATA[607,32] := 0.7355248;
   DATA[607,33] := 0.3063127;
   DATA[607,34] := 2.0;
   DATA[607,35] := 250.8331;
   DATA[607,36] := 1.649953;
   DATA[607,37] := 189.5988;
   DATA[607,38] := 0.000128152;
   DATA[607,39] := 1.0;
   DATA[608,0] := 2.620504;
   DATA[608,1] := 535.0936;
   DATA[608,2] := 2.0;
   DATA[608,3] := 2.0;
   DATA[608,4] := 262.1764;
   DATA[608,5] := 8.395475;
   DATA[608,6] := 327.8647;
   DATA[608,7] := 2.443341;
   DATA[608,8] := 2.0;
   DATA[608,9] := 2.0;
   DATA[608,10] := 2.0;
   DATA[608,11] := 19.69396;
   DATA[608,12] := 2.209653;
   DATA[608,13] := 986.4458;
   DATA[608,14] := 1.0;
   DATA[608,15] := 2.0;
   DATA[608,16] := 1.0;
   DATA[608,17] := 1.0;
   DATA[608,18] := 1.0;
   DATA[608,19] := 2.0;
   DATA[608,20] := 148.808;
   DATA[608,21] := 155.7806;
   DATA[608,22] := 1.719156;
   DATA[608,23] := 991.5535;
   DATA[608,24] := 2.0;
   DATA[608,25] := 2.0;
   DATA[608,26] := 7.880544;
   DATA[608,27] := 145.1679;
   DATA[608,28] := 263.4261;
   DATA[608,29] := 12.03538;
   DATA[608,30] := 1.724173;
   DATA[608,31] := 1.287691;
   DATA[608,32] := 0.7355248;
   DATA[608,33] := 0.306761;
   DATA[608,34] := 2.0;
   DATA[608,35] := 250.8331;
   DATA[608,36] := 1.649953;
   DATA[608,37] := 189.5988;
   DATA[608,38] := 0.000128152;
   DATA[608,39] := 1.0;
   DATA[609,0] := 2.649009;
   DATA[609,1] := 535.0936;
   DATA[609,2] := 2.0;
   DATA[609,3] := 2.0;
   DATA[609,4] := 262.1764;
   DATA[609,5] := 8.395475;
   DATA[609,6] := 327.8647;
   DATA[609,7] := 2.443597;
   DATA[609,8] := 2.0;
   DATA[609,9] := 2.0;
   DATA[609,10] := 2.0;
   DATA[609,11] := 19.69076;
   DATA[609,12] := 2.209653;
   DATA[609,13] := 986.4458;
   DATA[609,14] := 1.0;
   DATA[609,15] := 2.0;
   DATA[609,16] := 1.0;
   DATA[609,17] := 1.0;
   DATA[609,18] := 1.0;
   DATA[609,19] := 2.0;
   DATA[609,20] := 148.808;
   DATA[609,21] := 155.7806;
   DATA[609,22] := 1.719156;
   DATA[609,23] := 991.7073;
   DATA[609,24] := 2.0;
   DATA[609,25] := 2.0;
   DATA[609,26] := 7.880544;
   DATA[609,27] := 145.1679;
   DATA[609,28] := 263.4261;
   DATA[609,29] := 12.03538;
   DATA[609,30] := 1.725583;
   DATA[609,31] := 1.281158;
   DATA[609,32] := 0.7355248;
   DATA[609,33] := 0.306761;
   DATA[609,34] := 2.0;
   DATA[609,35] := 250.8331;
   DATA[609,36] := 1.649953;
   DATA[609,37] := 189.5988;
   DATA[609,38] := 0.000128152;
   DATA[609,39] := 1.0;
   DATA[610,0] := 2.668225;
   DATA[610,1] := 535.2899;
   DATA[610,2] := 2.0;
   DATA[610,3] := 2.0;
   DATA[610,4] := 262.1764;
   DATA[610,5] := 8.395475;
   DATA[610,6] := 327.8647;
   DATA[610,7] := 2.443597;
   DATA[610,8] := 2.0;
   DATA[610,9] := 2.0;
   DATA[610,10] := 2.0;
   DATA[610,11] := 19.69076;
   DATA[610,12] := 2.209653;
   DATA[610,13] := 986.1654;
   DATA[610,14] := 1.0;
   DATA[610,15] := 2.0;
   DATA[610,16] := 1.0;
   DATA[610,17] := 1.0;
   DATA[610,18] := 1.0;
   DATA[610,19] := 2.0;
   DATA[610,20] := 148.808;
   DATA[610,21] := 155.7806;
   DATA[610,22] := 1.717746;
   DATA[610,23] := 991.9764;
   DATA[610,24] := 2.0;
   DATA[610,25] := 2.0;
   DATA[610,26] := 7.880544;
   DATA[610,27] := 145.1679;
   DATA[610,28] := 263.4261;
   DATA[610,29] := 12.03538;
   DATA[610,30] := 1.725968;
   DATA[610,31] := 1.281158;
   DATA[610,32] := 0.7355248;
   DATA[610,33] := 0.306761;
   DATA[610,34] := 2.0;
   DATA[610,35] := 250.8331;
   DATA[610,36] := 1.649953;
   DATA[610,37] := 189.5988;
   DATA[610,38] := 0.000128152;
   DATA[610,39] := 1.0;
   DATA[611,0] := 2.668225;
   DATA[611,1] := 535.3291;
   DATA[611,2] := 2.0;
   DATA[611,3] := 2.0;
   DATA[611,4] := 262.1764;
   DATA[611,5] := 8.395475;
   DATA[611,6] := 327.8647;
   DATA[611,7] := 2.443597;
   DATA[611,8] := 2.0;
   DATA[611,9] := 2.0;
   DATA[611,10] := 2.0;
   DATA[611,11] := 19.72277;
   DATA[611,12] := 2.209653;
   DATA[611,13] := 986.2055;
   DATA[611,14] := 1.0;
   DATA[611,15] := 2.0;
   DATA[611,16] := 1.0;
   DATA[611,17] := 1.0;
   DATA[611,18] := 1.0;
   DATA[611,19] := 2.0;
   DATA[611,20] := 148.808;
   DATA[611,21] := 155.7806;
   DATA[611,22] := 1.716849;
   DATA[611,23] := 992.3994;
   DATA[611,24] := 2.0;
   DATA[611,25] := 2.0;
   DATA[611,26] := 7.880544;
   DATA[611,27] := 145.1679;
   DATA[611,28] := 263.3299;
   DATA[611,29] := 12.03538;
   DATA[611,30] := 1.726609;
   DATA[611,31] := 1.287947;
   DATA[611,32] := 0.7355248;
   DATA[611,33] := 0.306761;
   DATA[611,34] := 2.0;
   DATA[611,35] := 250.8331;
   DATA[611,36] := 1.649953;
   DATA[611,37] := 189.5988;
   DATA[611,38] := 0.000128152;
   DATA[611,39] := 1.0;
   DATA[612,0] := 2.644525;
   DATA[612,1] := 535.3291;
   DATA[612,2] := 2.0;
   DATA[612,3] := 2.0;
   DATA[612,4] := 262.1764;
   DATA[612,5] := 8.393232;
   DATA[612,6] := 327.8647;
   DATA[612,7] := 2.443597;
   DATA[612,8] := 2.0;
   DATA[612,9] := 2.0;
   DATA[612,10] := 2.0;
   DATA[612,11] := 19.72277;
   DATA[612,12] := 2.21119;
   DATA[612,13] := 986.2055;
   DATA[612,14] := 1.0;
   DATA[612,15] := 2.0;
   DATA[612,16] := 1.0;
   DATA[612,17] := 1.0;
   DATA[612,18] := 1.0;
   DATA[612,19] := 2.0;
   DATA[612,20] := 148.808;
   DATA[612,21] := 155.7806;
   DATA[612,22] := 1.716849;
   DATA[612,23] := 992.5916;
   DATA[612,24] := 2.0;
   DATA[612,25] := 2.0;
   DATA[612,26] := 7.880544;
   DATA[612,27] := 145.1679;
   DATA[612,28] := 263.3299;
   DATA[612,29] := 12.03538;
   DATA[612,30] := 1.727506;
   DATA[612,31] := 1.308441;
   DATA[612,32] := 0.7355248;
   DATA[612,33] := 0.306761;
   DATA[612,34] := 2.0;
   DATA[612,35] := 250.9933;
   DATA[612,36] := 1.649953;
   DATA[612,37] := 189.8231;
   DATA[612,38] := 0.000128152;
   DATA[612,39] := 1.0;
   DATA[613,0] := 2.624347;
   DATA[613,1] := 535.2899;
   DATA[613,2] := 2.0;
   DATA[613,3] := 2.0;
   DATA[613,4] := 262.1764;
   DATA[613,5] := 8.393232;
   DATA[613,6] := 327.8647;
   DATA[613,7] := 2.443725;
   DATA[613,8] := 2.0;
   DATA[613,9] := 2.0;
   DATA[613,10] := 2.0;
   DATA[613,11] := 19.72277;
   DATA[613,12] := 2.21119;
   DATA[613,13] := 985.8851;
   DATA[613,14] := 1.0;
   DATA[613,15] := 2.0;
   DATA[613,16] := 1.0;
   DATA[613,17] := 1.0;
   DATA[613,18] := 1.0;
   DATA[613,19] := 2.0;
   DATA[613,20] := 148.808;
   DATA[613,21] := 155.7806;
   DATA[613,22] := 1.716849;
   DATA[613,23] := 992.5147;
   DATA[613,24] := 2.0;
   DATA[613,25] := 2.0;
   DATA[613,26] := 7.880544;
   DATA[613,27] := 145.1679;
   DATA[613,28] := 263.1697;
   DATA[613,29] := 12.03538;
   DATA[613,30] := 1.727506;
   DATA[613,31] := 1.312412;
   DATA[613,32] := 0.7355248;
   DATA[613,33] := 0.306761;
   DATA[613,34] := 2.0;
   DATA[613,35] := 250.9933;
   DATA[613,36] := 1.649953;
   DATA[613,37] := 189.9353;
   DATA[613,38] := 0.000128152;
   DATA[613,39] := 1.0;
   DATA[614,0] := 2.620824;
   DATA[614,1] := 535.2506;
   DATA[614,2] := 2.0;
   DATA[614,3] := 2.0;
   DATA[614,4] := 262.1764;
   DATA[614,5] := 8.393232;
   DATA[614,6] := 327.8647;
   DATA[614,7] := 2.443725;
   DATA[614,8] := 2.0;
   DATA[614,9] := 2.0;
   DATA[614,10] := 2.0;
   DATA[614,11] := 19.72277;
   DATA[614,12] := 2.21119;
   DATA[614,13] := 985.845;
   DATA[614,14] := 1.0;
   DATA[614,15] := 2.0;
   DATA[614,16] := 1.0;
   DATA[614,17] := 1.0;
   DATA[614,18] := 1.0;
   DATA[614,19] := 2.0;
   DATA[614,20] := 148.808;
   DATA[614,21] := 155.7806;
   DATA[614,22] := 1.716849;
   DATA[614,23] := 992.2841;
   DATA[614,24] := 2.0;
   DATA[614,25] := 2.0;
   DATA[614,26] := 7.880544;
   DATA[614,27] := 145.1679;
   DATA[614,28] := 263.1697;
   DATA[614,29] := 12.03538;
   DATA[614,30] := 1.729813;
   DATA[614,31] := 1.330601;
   DATA[614,32] := 0.7355248;
   DATA[614,33] := 0.306761;
   DATA[614,34] := 2.0;
   DATA[614,35] := 251.0734;
   DATA[614,36] := 1.649953;
   DATA[614,37] := 189.9353;
   DATA[614,38] := 0.000128152;
   DATA[614,39] := 1.0;
   DATA[615,0] := 2.617622;
   DATA[615,1] := 535.4469;
   DATA[615,2] := 2.0;
   DATA[615,3] := 2.0;
   DATA[615,4] := 262.1764;
   DATA[615,5] := 8.394514;
   DATA[615,6] := 327.8647;
   DATA[615,7] := 2.443725;
   DATA[615,8] := 2.0;
   DATA[615,9] := 2.0;
   DATA[615,10] := 2.0;
   DATA[615,11] := 19.72277;
   DATA[615,12] := 2.21119;
   DATA[615,13] := 986.2455;
   DATA[615,14] := 1.0;
   DATA[615,15] := 2.0;
   DATA[615,16] := 1.0;
   DATA[615,17] := 1.0;
   DATA[615,18] := 1.0;
   DATA[615,19] := 2.0;
   DATA[615,20] := 148.808;
   DATA[615,21] := 155.7806;
   DATA[615,22] := 1.716849;
   DATA[615,23] := 992.2841;
   DATA[615,24] := 2.0;
   DATA[615,25] := 2.0;
   DATA[615,26] := 7.880544;
   DATA[615,27] := 145.1679;
   DATA[615,28] := 263.1377;
   DATA[615,29] := 12.03538;
   DATA[615,30] := 1.729813;
   DATA[615,31] := 1.326502;
   DATA[615,32] := 0.7355248;
   DATA[615,33] := 0.306761;
   DATA[615,34] := 2.0;
   DATA[615,35] := 251.2817;
   DATA[615,36] := 1.649953;
   DATA[615,37] := 189.9353;
   DATA[615,38] := 0.000128152;
   DATA[615,39] := 1.0;
   DATA[616,0] := 2.596163;
   DATA[616,1] := 535.4861;
   DATA[616,2] := 2.0;
   DATA[616,3] := 2.0;
   DATA[616,4] := 262.1764;
   DATA[616,5] := 8.394514;
   DATA[616,6] := 327.8647;
   DATA[616,7] := 2.44206;
   DATA[616,8] := 2.0;
   DATA[616,9] := 2.0;
   DATA[616,10] := 2.0;
   DATA[616,11] := 19.72277;
   DATA[616,12] := 2.21119;
   DATA[616,13] := 986.0453;
   DATA[616,14] := 1.0;
   DATA[616,15] := 2.0;
   DATA[616,16] := 1.0;
   DATA[616,17] := 1.0;
   DATA[616,18] := 1.0;
   DATA[616,19] := 2.0;
   DATA[616,20] := 148.808;
   DATA[616,21] := 155.7806;
   DATA[616,22] := 1.717489;
   DATA[616,23] := 992.1687;
   DATA[616,24] := 2.0;
   DATA[616,25] := 2.0;
   DATA[616,26] := 7.880544;
   DATA[616,27] := 145.1679;
   DATA[616,28] := 263.1377;
   DATA[616,29] := 12.03538;
   DATA[616,30] := 1.729813;
   DATA[616,31] := 1.312668;
   DATA[616,32] := 0.7355248;
   DATA[616,33] := 0.306761;
   DATA[616,34] := 2.0;
   DATA[616,35] := 251.2817;
   DATA[616,36] := 1.730048;
   DATA[616,37] := 189.9353;
   DATA[616,38] := 0.000128152;
   DATA[616,39] := 1.0;
   DATA[617,0] := 2.585594;
   DATA[617,1] := 535.3291;
   DATA[617,2] := 2.0;
   DATA[617,3] := 2.0;
   DATA[617,4] := 262.1764;
   DATA[617,5] := 8.394514;
   DATA[617,6] := 327.8647;
   DATA[617,7] := 2.439496;
   DATA[617,8] := 2.0;
   DATA[617,9] := 2.0;
   DATA[617,10] := 2.0;
   DATA[617,11] := 19.66195;
   DATA[617,12] := 2.21119;
   DATA[617,13] := 986.0052;
   DATA[617,14] := 1.0;
   DATA[617,15] := 2.0;
   DATA[617,16] := 1.0;
   DATA[617,17] := 1.0;
   DATA[617,18] := 1.0;
   DATA[617,19] := 2.0;
   DATA[617,20] := 148.808;
   DATA[617,21] := 155.7806;
   DATA[617,22] := 1.717489;
   DATA[617,23] := 992.3994;
   DATA[617,24] := 2.0;
   DATA[617,25] := 2.0;
   DATA[617,26] := 7.880544;
   DATA[617,27] := 145.1679;
   DATA[617,28] := 263.1377;
   DATA[617,29] := 12.03538;
   DATA[617,30] := 1.729813;
   DATA[617,31] := 1.302037;
   DATA[617,32] := 0.7355248;
   DATA[617,33] := 0.306761;
   DATA[617,34] := 2.0;
   DATA[617,35] := 251.2817;
   DATA[617,36] := 1.730048;
   DATA[617,37] := 189.9353;
   DATA[617,38] := 0.000128152;
   DATA[617,39] := 1.0;
   DATA[618,0] := 2.563174;
   DATA[618,1] := 535.6431;
   DATA[618,2] := 2.0;
   DATA[618,3] := 2.0;
   DATA[618,4] := 262.1764;
   DATA[618,5] := 8.394514;
   DATA[618,6] := 327.8647;
   DATA[618,7] := 2.439496;
   DATA[618,8] := 2.0;
   DATA[618,9] := 2.0;
   DATA[618,10] := 2.0;
   DATA[618,11] := 19.66195;
   DATA[618,12] := 2.21119;
   DATA[618,13] := 985.7649;
   DATA[618,14] := 1.0;
   DATA[618,15] := 2.0;
   DATA[618,16] := 1.0;
   DATA[618,17] := 1.0;
   DATA[618,18] := 1.0;
   DATA[618,19] := 2.0;
   DATA[618,20] := 148.808;
   DATA[618,21] := 155.7806;
   DATA[618,22] := 1.719924;
   DATA[618,23] := 992.361;
   DATA[618,24] := 2.0;
   DATA[618,25] := 2.0;
   DATA[618,26] := 7.880544;
   DATA[618,27] := 145.1679;
   DATA[618,28] := 263.1377;
   DATA[618,29] := 12.03538;
   DATA[618,30] := 1.729813;
   DATA[618,31] := 1.291405;
   DATA[618,32] := 0.7355248;
   DATA[618,33] := 0.306761;
   DATA[618,34] := 2.0;
   DATA[618,35] := 251.2817;
   DATA[618,36] := 1.730048;
   DATA[618,37] := 189.9353;
   DATA[618,38] := 0.000128152;
   DATA[618,39] := 1.0;
   DATA[619,0] := 2.547481;
   DATA[619,1] := 535.9179;
   DATA[619,2] := 2.0;
   DATA[619,3] := 2.0;
   DATA[619,4] := 262.1764;
   DATA[619,5] := 8.394514;
   DATA[619,6] := 327.8647;
   DATA[619,7] := 2.439496;
   DATA[619,8] := 2.0;
   DATA[619,9] := 2.0;
   DATA[619,10] := 2.0;
   DATA[619,11] := 19.66195;
   DATA[619,12] := 2.21119;
   DATA[619,13] := 985.6848;
   DATA[619,14] := 1.0;
   DATA[619,15] := 2.0;
   DATA[619,16] := 1.0;
   DATA[619,17] := 1.0;
   DATA[619,18] := 1.0;
   DATA[619,19] := 2.0;
   DATA[619,20] := 148.808;
   DATA[619,21] := 155.7806;
   DATA[619,22] := 1.719924;
   DATA[619,23] := 992.6685;
   DATA[619,24] := 2.0;
   DATA[619,25] := 2.0;
   DATA[619,26] := 7.880544;
   DATA[619,27] := 145.1166;
   DATA[619,28] := 263.1377;
   DATA[619,29] := 12.03538;
   DATA[619,30] := 1.729813;
   DATA[619,31] := 1.280261;
   DATA[619,32] := 0.7355248;
   DATA[619,33] := 0.306761;
   DATA[619,34] := 2.0;
   DATA[619,35] := 251.1215;
   DATA[619,36] := 1.730048;
   DATA[619,37] := 189.9353;
   DATA[619,38] := 0.000128152;
   DATA[619,39] := 1.0;
   DATA[620,0] := 2.525702;
   DATA[620,1] := 536.2712;
   DATA[620,2] := 2.0;
   DATA[620,3] := 2.0;
   DATA[620,4] := 262.1764;
   DATA[620,5] := 8.394514;
   DATA[620,6] := 327.8647;
   DATA[620,7] := 2.439496;
   DATA[620,8] := 2.0;
   DATA[620,9] := 2.0;
   DATA[620,10] := 2.0;
   DATA[620,11] := 19.66195;
   DATA[620,12] := 2.21119;
   DATA[620,13] := 985.4044;
   DATA[620,14] := 1.0;
   DATA[620,15] := 2.0;
   DATA[620,16] := 1.0;
   DATA[620,17] := 1.0;
   DATA[620,18] := 1.0;
   DATA[620,19] := 2.0;
   DATA[620,20] := 148.808;
   DATA[620,21] := 155.7806;
   DATA[620,22] := 1.719924;
   DATA[620,23] := 992.8992;
   DATA[620,24] := 2.0;
   DATA[620,25] := 2.0;
   DATA[620,26] := 7.880544;
   DATA[620,27] := 145.1166;
   DATA[620,28] := 263.1377;
   DATA[620,29] := 12.03538;
   DATA[620,30] := 1.729813;
   DATA[620,31] := 1.271679;
   DATA[620,32] := 0.7355248;
   DATA[620,33] := 0.306761;
   DATA[620,34] := 2.0;
   DATA[620,35] := 251.1215;
   DATA[620,36] := 1.730048;
   DATA[620,37] := 189.8552;
   DATA[620,38] := 0.000128152;
   DATA[620,39] := 1.0;
   DATA[621,0] := 2.510649;
   DATA[621,1] := 536.4675;
   DATA[621,2] := 2.0;
   DATA[621,3] := 2.0;
   DATA[621,4] := 262.1764;
   DATA[621,5] := 8.394514;
   DATA[621,6] := 327.8647;
   DATA[621,7] := 2.441419;
   DATA[621,8] := 2.0;
   DATA[621,9] := 2.0;
   DATA[621,10] := 2.0;
   DATA[621,11] := 19.71637;
   DATA[621,12] := 2.210166;
   DATA[621,13] := 985.8049;
   DATA[621,14] := 1.0;
   DATA[621,15] := 2.0;
   DATA[621,16] := 1.0;
   DATA[621,17] := 1.0;
   DATA[621,18] := 1.0;
   DATA[621,19] := 2.0;
   DATA[621,20] := 148.808;
   DATA[621,21] := 155.7806;
   DATA[621,22] := 1.719924;
   DATA[621,23] := 992.8992;
   DATA[621,24] := 2.0;
   DATA[621,25] := 2.0;
   DATA[621,26] := 7.880544;
   DATA[621,27] := 145.1166;
   DATA[621,28] := 263.1377;
   DATA[621,29] := 12.03538;
   DATA[621,30] := 1.729813;
   DATA[621,31] := 1.271679;
   DATA[621,32] := 0.7355248;
   DATA[621,33] := 0.306761;
   DATA[621,34] := 2.0;
   DATA[621,35] := 251.1215;
   DATA[621,36] := 1.601897;
   DATA[621,37] := 189.8552;
   DATA[621,38] := 0.000128152;
   DATA[621,39] := 1.0;
   DATA[622,0] := 2.491112;
   DATA[622,1] := 536.6637;
   DATA[622,2] := 2.0;
   DATA[622,3] := 2.0;
   DATA[622,4] := 262.1764;
   DATA[622,5] := 8.394514;
   DATA[622,6] := 327.8647;
   DATA[622,7] := 2.441803;
   DATA[622,8] := 2.0;
   DATA[622,9] := 2.0;
   DATA[622,10] := 2.0;
   DATA[622,11] := 19.71637;
   DATA[622,12] := 2.209397;
   DATA[622,13] := 985.7649;
   DATA[622,14] := 1.0;
   DATA[622,15] := 2.0;
   DATA[622,16] := 1.0;
   DATA[622,17] := 1.0;
   DATA[622,18] := 1.0;
   DATA[622,19] := 2.0;
   DATA[622,20] := 148.808;
   DATA[622,21] := 155.7806;
   DATA[622,22] := 1.718771;
   DATA[622,23] := 992.7454;
   DATA[622,24] := 2.0;
   DATA[622,25] := 2.0;
   DATA[622,26] := 7.880544;
   DATA[622,27] := 145.1166;
   DATA[622,28] := 263.1377;
   DATA[622,29] := 12.03538;
   DATA[622,30] := 1.729813;
   DATA[622,31] := 1.261816;
   DATA[622,32] := 0.7355248;
   DATA[622,33] := 0.3075937;
   DATA[622,34] := 2.0;
   DATA[622,35] := 251.1215;
   DATA[622,36] := 1.601897;
   DATA[622,37] := 189.8552;
   DATA[622,38] := 0.000128152;
   DATA[622,39] := 1.0;
   DATA[623,0] := 2.491112;
   DATA[623,1] := 536.6637;
   DATA[623,2] := 2.0;
   DATA[623,3] := 2.0;
   DATA[623,4] := 262.1764;
   DATA[623,5] := 8.394514;
   DATA[623,6] := 327.8647;
   DATA[623,7] := 2.441803;
   DATA[623,8] := 2.0;
   DATA[623,9] := 2.0;
   DATA[623,10] := 2.0;
   DATA[623,11] := 19.71637;
   DATA[623,12] := 2.209397;
   DATA[623,13] := 985.7649;
   DATA[623,14] := 1.0;
   DATA[623,15] := 2.0;
   DATA[623,16] := 1.0;
   DATA[623,17] := 1.0;
   DATA[623,18] := 1.0;
   DATA[623,19] := 2.0;
   DATA[623,20] := 148.808;
   DATA[623,21] := 155.7806;
   DATA[623,22] := 1.718771;
   DATA[623,23] := 992.7454;
   DATA[623,24] := 2.0;
   DATA[623,25] := 2.0;
   DATA[623,26] := 7.880544;
   DATA[623,27] := 145.1166;
   DATA[623,28] := 263.1377;
   DATA[623,29] := 12.03538;
   DATA[623,30] := 1.729813;
   DATA[623,31] := 1.261816;
   DATA[623,32] := 0.7355248;
   DATA[623,33] := 0.3075937;
   DATA[623,34] := 2.0;
   DATA[623,35] := 251.1215;
   DATA[623,36] := 1.601897;
   DATA[623,37] := 189.8552;
   DATA[623,38] := 0.000128152;
   DATA[623,39] := 1.0;
   DATA[624,0] := 2.477661;
   DATA[624,1] := 536.6245;
   DATA[624,2] := 2.0;
   DATA[624,3] := 2.0;
   DATA[624,4] := 262.1764;
   DATA[624,5] := 8.394514;
   DATA[624,6] := 327.8647;
   DATA[624,7] := 2.441803;
   DATA[624,8] := 2.0;
   DATA[624,9] := 2.0;
   DATA[624,10] := 2.0;
   DATA[624,11] := 19.71637;
   DATA[624,12] := 2.209397;
   DATA[624,13] := 985.4845;
   DATA[624,14] := 1.0;
   DATA[624,15] := 2.0;
   DATA[624,16] := 1.0;
   DATA[624,17] := 1.0;
   DATA[624,18] := 1.0;
   DATA[624,19] := 2.0;
   DATA[624,20] := 148.808;
   DATA[624,21] := 155.7806;
   DATA[624,22] := 1.717105;
   DATA[624,23] := 992.7454;
   DATA[624,24] := 2.0;
   DATA[624,25] := 2.0;
   DATA[624,26] := 7.880544;
   DATA[624,27] := 145.1166;
   DATA[624,28] := 263.1377;
   DATA[624,29] := 12.03538;
   DATA[624,30] := 1.729813;
   DATA[624,31] := 1.261048;
   DATA[624,32] := 0.7355248;
   DATA[624,33] := 0.3084265;
   DATA[624,34] := 2.0;
   DATA[624,35] := 251.1215;
   DATA[624,36] := 1.601897;
   DATA[624,37] := 189.8552;
   DATA[624,38] := 0.000128152;
   DATA[624,39] := 1.0;
   DATA[625,0] := 2.460045;
   DATA[625,1] := 536.8207;
   DATA[625,2] := 2.0;
   DATA[625,3] := 2.0;
   DATA[625,4] := 262.1764;
   DATA[625,5] := 8.394514;
   DATA[625,6] := 327.8647;
   DATA[625,7] := 2.440393;
   DATA[625,8] := 2.0;
   DATA[625,9] := 2.0;
   DATA[625,10] := 2.0;
   DATA[625,11] := 19.70357;
   DATA[625,12] := 2.209397;
   DATA[625,13] := 985.6848;
   DATA[625,14] := 1.0;
   DATA[625,15] := 2.0;
   DATA[625,16] := 1.0;
   DATA[625,17] := 1.0;
   DATA[625,18] := 1.0;
   DATA[625,19] := 2.0;
   DATA[625,20] := 148.808;
   DATA[625,21] := 155.7806;
   DATA[625,22] := 1.717105;
   DATA[625,23] := 992.7454;
   DATA[625,24] := 2.0;
   DATA[625,25] := 2.0;
   DATA[625,26] := 7.880544;
   DATA[625,27] := 145.1166;
   DATA[625,28] := 263.1377;
   DATA[625,29] := 12.03538;
   DATA[625,30] := 1.728916;
   DATA[625,31] := 1.261048;
   DATA[625,32] := 0.7355248;
   DATA[625,33] := 0.3084265;
   DATA[625,34] := 2.0;
   DATA[625,35] := 250.8972;
   DATA[625,36] := 1.69801;
   DATA[625,37] := 189.6469;
   DATA[625,38] := 0.000128152;
   DATA[625,39] := 1.0;
   DATA[626,0] := 2.447234;
   DATA[626,1] := 536.86;
   DATA[626,2] := 2.0;
   DATA[626,3] := 2.0;
   DATA[626,4] := 262.1764;
   DATA[626,5] := 8.394514;
   DATA[626,6] := 327.8647;
   DATA[626,7] := 2.439625;
   DATA[626,8] := 2.0;
   DATA[626,9] := 2.0;
   DATA[626,10] := 2.0;
   DATA[626,11] := 19.68756;
   DATA[626,12] := 2.209397;
   DATA[626,13] := 985.6848;
   DATA[626,14] := 1.0;
   DATA[626,15] := 2.0;
   DATA[626,16] := 1.0;
   DATA[626,17] := 1.0;
   DATA[626,18] := 1.0;
   DATA[626,19] := 2.0;
   DATA[626,20] := 148.808;
   DATA[626,21] := 155.7806;
   DATA[626,22] := 1.717105;
   DATA[626,23] := 992.2841;
   DATA[626,24] := 2.0;
   DATA[626,25] := 2.0;
   DATA[626,26] := 7.880544;
   DATA[626,27] := 145.1166;
   DATA[626,28] := 263.1377;
   DATA[626,29] := 12.03538;
   DATA[626,30] := 1.726865;
   DATA[626,31] := 1.272064;
   DATA[626,32] := 0.7355248;
   DATA[626,33] := 0.3084265;
   DATA[626,34] := 2.0;
   DATA[626,35] := 250.8972;
   DATA[626,36] := 1.69801;
   DATA[626,37] := 189.5027;
   DATA[626,38] := 0.000128152;
   DATA[626,39] := 1.0;
   DATA[627,0] := 2.431861;
   DATA[627,1] := 536.9777;
   DATA[627,2] := 2.0;
   DATA[627,3] := 2.0;
   DATA[627,4] := 262.1764;
   DATA[627,5] := 8.394514;
   DATA[627,6] := 327.8647;
   DATA[627,7] := 2.439625;
   DATA[627,8] := 2.0;
   DATA[627,9] := 2.0;
   DATA[627,10] := 2.0;
   DATA[627,11] := 19.68756;
   DATA[627,12] := 2.209397;
   DATA[627,13] := 985.5646;
   DATA[627,14] := 1.0;
   DATA[627,15] := 2.0;
   DATA[627,16] := 1.0;
   DATA[627,17] := 1.0;
   DATA[627,18] := 1.0;
   DATA[627,19] := 2.0;
   DATA[627,20] := 148.808;
   DATA[627,21] := 155.7806;
   DATA[627,22] := 1.717105;
   DATA[627,23] := 992.3994;
   DATA[627,24] := 2.0;
   DATA[627,25] := 2.0;
   DATA[627,26] := 7.880544;
   DATA[627,27] := 145.1166;
   DATA[627,28] := 263.1377;
   DATA[627,29] := 12.03538;
   DATA[627,30] := 1.726865;
   DATA[627,31] := 1.287306;
   DATA[627,32] := 0.7355248;
   DATA[627,33] := 0.3084265;
   DATA[627,34] := 2.0;
   DATA[627,35] := 250.8972;
   DATA[627,36] := 1.69801;
   DATA[627,37] := 189.5027;
   DATA[627,38] := 0.000128152;
   DATA[627,39] := 1.0;
   DATA[628,0] := 2.431861;
   DATA[628,1] := 536.6637;
   DATA[628,2] := 2.0;
   DATA[628,3] := 2.0;
   DATA[628,4] := 262.1764;
   DATA[628,5] := 8.394514;
   DATA[628,6] := 327.7621;
   DATA[628,7] := 2.439625;
   DATA[628,8] := 2.0;
   DATA[628,9] := 2.0;
   DATA[628,10] := 2.0;
   DATA[628,11] := 19.68756;
   DATA[628,12] := 2.206707;
   DATA[628,13] := 985.4845;
   DATA[628,14] := 1.0;
   DATA[628,15] := 2.0;
   DATA[628,16] := 1.0;
   DATA[628,17] := 1.0;
   DATA[628,18] := 1.0;
   DATA[628,19] := 2.0;
   DATA[628,20] := 148.808;
   DATA[628,21] := 155.7806;
   DATA[628,22] := 1.717105;
   DATA[628,23] := 992.361;
   DATA[628,24] := 2.0;
   DATA[628,25] := 2.0;
   DATA[628,26] := 7.880544;
   DATA[628,27] := 145.1166;
   DATA[628,28] := 263.1377;
   DATA[628,29] := 12.03538;
   DATA[628,30] := 1.726865;
   DATA[628,31] := 1.300756;
   DATA[628,32] := 0.7355248;
   DATA[628,33] := 0.3084265;
   DATA[628,34] := 2.0;
   DATA[628,35] := 250.8972;
   DATA[628,36] := 1.69801;
   DATA[628,37] := 189.5027;
   DATA[628,38] := 0.000128152;
   DATA[628,39] := 1.0;
   DATA[629,0] := 2.451398;
   DATA[629,1] := 536.2319;
   DATA[629,2] := 2.0;
   DATA[629,3] := 2.0;
   DATA[629,4] := 262.1764;
   DATA[629,5] := 8.394514;
   DATA[629,6] := 327.7621;
   DATA[629,7] := 2.439625;
   DATA[629,8] := 2.0;
   DATA[629,9] := 2.0;
   DATA[629,10] := 2.0;
   DATA[629,11] := 19.68756;
   DATA[629,12] := 2.206707;
   DATA[629,13] := 985.4445;
   DATA[629,14] := 1.0;
   DATA[629,15] := 2.0;
   DATA[629,16] := 1.0;
   DATA[629,17] := 1.0;
   DATA[629,18] := 1.0;
   DATA[629,19] := 2.0;
   DATA[629,20] := 148.808;
   DATA[629,21] := 155.7806;
   DATA[629,22] := 1.717105;
   DATA[629,23] := 992.6685;
   DATA[629,24] := 2.0;
   DATA[629,25] := 2.0;
   DATA[629,26] := 7.880544;
   DATA[629,27] := 145.1166;
   DATA[629,28] := 263.1377;
   DATA[629,29] := 12.03538;
   DATA[629,30] := 1.726865;
   DATA[629,31] := 1.302037;
   DATA[629,32] := 0.7355248;
   DATA[629,33] := 0.3084265;
   DATA[629,34] := 2.0;
   DATA[629,35] := 250.8972;
   DATA[629,36] := 1.69801;
   DATA[629,37] := 189.5027;
   DATA[629,38] := 0.000128152;
   DATA[629,39] := 1.0;
   DATA[630,0] := 2.507126;
   DATA[630,1] := 536.0749;
   DATA[630,2] := 2.0;
   DATA[630,3] := 2.0;
   DATA[630,4] := 262.1764;
   DATA[630,5] := 8.396116;
   DATA[630,6] := 327.7621;
   DATA[630,7] := 2.439625;
   DATA[630,8] := 2.0;
   DATA[630,9] := 2.0;
   DATA[630,10] := 2.0;
   DATA[630,11] := 19.65235;
   DATA[630,12] := 2.209653;
   DATA[630,13] := 985.4845;
   DATA[630,14] := 1.0;
   DATA[630,15] := 2.0;
   DATA[630,16] := 1.0;
   DATA[630,17] := 1.0;
   DATA[630,18] := 1.0;
   DATA[630,19] := 2.0;
   DATA[630,20] := 148.808;
   DATA[630,21] := 155.7806;
   DATA[630,22] := 1.717105;
   DATA[630,23] := 992.6685;
   DATA[630,24] := 2.0;
   DATA[630,25] := 2.0;
   DATA[630,26] := 7.878621;
   DATA[630,27] := 145.1166;
   DATA[630,28] := 263.1377;
   DATA[630,29] := 12.03538;
   DATA[630,30] := 1.7293;
   DATA[630,31] := 1.302037;
   DATA[630,32] := 0.7355248;
   DATA[630,33] := 0.3084265;
   DATA[630,34] := 2.0;
   DATA[630,35] := 250.8972;
   DATA[630,36] := 1.69801;
   DATA[630,37] := 189.6148;
   DATA[630,38] := 0.000128152;
   DATA[630,39] := 1.0;
   DATA[631,0] := 2.53467;
   DATA[631,1] := 535.4076;
   DATA[631,2] := 2.0;
   DATA[631,3] := 2.0;
   DATA[631,4] := 262.1764;
   DATA[631,5] := 8.396116;
   DATA[631,6] := 327.7621;
   DATA[631,7] := 2.439625;
   DATA[631,8] := 2.0;
   DATA[631,9] := 2.0;
   DATA[631,10] := 2.0;
   DATA[631,11] := 19.65235;
   DATA[631,12] := 2.209653;
   DATA[631,13] := 985.5646;
   DATA[631,14] := 1.0;
   DATA[631,15] := 2.0;
   DATA[631,16] := 1.0;
   DATA[631,17] := 1.0;
   DATA[631,18] := 1.0;
   DATA[631,19] := 2.0;
   DATA[631,20] := 148.808;
   DATA[631,21] := 155.7806;
   DATA[631,22] := 1.717105;
   DATA[631,23] := 992.7454;
   DATA[631,24] := 2.0;
   DATA[631,25] := 2.0;
   DATA[631,26] := 7.87798;
   DATA[631,27] := 145.1166;
   DATA[631,28] := 263.1377;
   DATA[631,29] := 12.03538;
   DATA[631,30] := 1.7293;
   DATA[631,31] := 1.301012;
   DATA[631,32] := 0.7355248;
   DATA[631,33] := 0.3084265;
   DATA[631,34] := 2.0;
   DATA[631,35] := 250.8972;
   DATA[631,36] := 1.69801;
   DATA[631,37] := 189.6148;
   DATA[631,38] := 0.000128152;
   DATA[631,39] := 1.0;
   DATA[632,0] := 2.578868;
   DATA[632,1] := 535.1329;
   DATA[632,2] := 2.0;
   DATA[632,3] := 2.0;
   DATA[632,4] := 262.1764;
   DATA[632,5] := 8.396116;
   DATA[632,6] := 327.7621;
   DATA[632,7] := 2.441675;
   DATA[632,8] := 2.0;
   DATA[632,9] := 2.0;
   DATA[632,10] := 2.0;
   DATA[632,11] := 19.68756;
   DATA[632,12] := 2.209653;
   DATA[632,13] := 985.6047;
   DATA[632,14] := 1.0;
   DATA[632,15] := 2.0;
   DATA[632,16] := 1.0;
   DATA[632,17] := 1.0;
   DATA[632,18] := 1.0;
   DATA[632,19] := 2.0;
   DATA[632,20] := 148.808;
   DATA[632,21] := 155.7806;
   DATA[632,22] := 1.719156;
   DATA[632,23] := 992.361;
   DATA[632,24] := 2.0;
   DATA[632,25] := 2.0;
   DATA[632,26] := 7.87798;
   DATA[632,27] := 145.1166;
   DATA[632,28] := 263.1377;
   DATA[632,29] := 12.03538;
   DATA[632,30] := 1.731095;
   DATA[632,31] := 1.282439;
   DATA[632,32] := 0.7355248;
   DATA[632,33] := 0.3084265;
   DATA[632,34] := 2.0;
   DATA[632,35] := 250.8972;
   DATA[632,36] := 1.69801;
   DATA[632,37] := 189.6148;
   DATA[632,38] := 0.000128152;
   DATA[632,39] := 1.0;
   DATA[633,0] := 2.608334;
   DATA[633,1] := 534.7403;
   DATA[633,2] := 2.0;
   DATA[633,3] := 2.0;
   DATA[633,4] := 262.1764;
   DATA[633,5] := 8.396116;
   DATA[633,6] := 327.7621;
   DATA[633,7] := 2.441675;
   DATA[633,8] := 2.0;
   DATA[633,9] := 2.0;
   DATA[633,10] := 2.0;
   DATA[633,11] := 19.68756;
